//     Term 27 (AT2000-0250)/CC Outputs/Current setpoint value Ch.11 <-> Data Pointer/CurrentSetpointValues[10]
//     Term 27 (AT2000-0250)/CC Outputs/Current setpoint value Ch.12 <-> Data Pointer/CurrentSetpointValues[11]
//     Term 27 (AT2000-0250)/CC Outputs/Current setpoint value Ch.13 <-> Data Pointer/CurrentSetpointValues[12]
//     Term 27 (AT2000-0250)/CC Outputs/Current setpoint value Ch.14 <-> Data Pointer/CurrentSetpointValues[13]
//     Term 27 (AT2000-0250)/CC Outputs/Current setpoint value Ch.15 <-> Data Pointer/CurrentSetpointValues[14]
//     Term 27 (AT2000-0250)/CC Outputs/Current setpoint value Ch.2 <-> Data Pointer/CurrentSetpointValues[1]
//     Term 27 (AT2000-0250)/CC Outputs/Current setpoint value Ch.3 <-> Data Pointer/CurrentSetpointValues[2]
//     Term 27 (AT2000-0250)/CC Outputs/Current setpoint value Ch.4 <-> Data Pointer/CurrentSetpointValues[3]
//     Term 27 (AT2000-0250)/CC Outputs/Current setpoint value Ch.5 <-> Data Pointer/CurrentSetpointValues[4]
//     Term 27 (AT2000-0250)/CC Outputs/Current setpoint value Ch.6 <-> Data Pointer/CurrentSetpointValues[5]
//     Term 27 (AT2000-0250)/CC Outputs/Current setpoint value Ch.7 <-> Data Pointer/CurrentSetpointValues[6]
//     Term 27 (AT2000-0250)/CC Outputs/Current setpoint value Ch.8 <-> Data Pointer/CurrentSetpointValues[7]
//     Term 27 (AT2000-0250)/CC Outputs/Current setpoint value Ch.9 <-> Data Pointer/CurrentSetpointValues[8]
//     Term 27 (AT2000-0250)/Term 28 (AT2000-5250)/FB Inputs/Value Channel 01 <-> Data Pointer/RawPositionValues[0]
//     Term 27 (AT2000-0250)/Term 28 (AT2000-5250)/FB Inputs/Value Channel 02 <-> Data Pointer/RawPositionValues[1]
//     Term 27 (AT2000-0250)/Term 28 (AT2000-5250)/FB Inputs/Value Channel 03 <-> Data Pointer/RawPositionValues[2]
//     Term 27 (AT2000-0250)/Term 28 (AT2000-5250)/FB Inputs/Value Channel 04 <-> Data Pointer/RawPositionValues[3]
//     Term 27 (AT2000-0250)/Term 28 (AT2000-5250)/FB Inputs/Value Channel 05 <-> Data Pointer/RawPositionValues[4]
//     Term 27 (AT2000-0250)/Term 28 (AT2000-5250)/FB Inputs/Value Channel 06 <-> Data Pointer/RawPositionValues[5]
//     Term 27 (AT2000-0250)/Term 28 (AT2000-5250)/FB Inputs/Value Channel 07 <-> Data Pointer/RawPositionValues[6]
//     Term 27 (AT2000-0250)/Term 28 (AT2000-5250)/FB Inputs/Value Channel 08 <-> Data Pointer/RawPositionValues[7]
//     Term 27 (AT2000-0250)/Term 28 (AT2000-5250)/FB Inputs/Value Channel 09 <-> Data Pointer/RawPositionValues[8]
//     Term 27 (AT2000-0250)/Term 28 (AT2000-5250)/FB Inputs/Value Channel 10 <-> Data Pointer/RawPositionValues[9]
//     Term 27 (AT2000-0250)/Term 28 (AT2000-5250)/FB Inputs/Value Channel 11 <-> Data Pointer/RawPositionValues[10]
//     Term 27 (AT2000-0250)/Term 28 (AT2000-5250)/FB Inputs/Value Channel 12 <-> Data Pointer/RawPositionValues[11]
//     Term 27 (AT2000-0250)/Term 28 (AT2000-5250)/FB Inputs/Value Channel 13 <-> Data Pointer/RawPositionValues[12]
//     Term 27 (AT2000-0250)/Term 28 (AT2000-5250)/FB Inputs/Value Channel 14 <-> Data Pointer/RawPositionValues[13]
//     Term 27 (AT2000-0250)/Term 28 (AT2000-5250)/FB Inputs/Value Channel 15 <-> Data Pointer/RawPositionValues[14]
//     Term 27 (AT2000-0250)/Term 28 (AT2000-5250)/FB Inputs/Value Channel 16 <-> Data Pointer/RawPositionValues[15]
//     Term 27 (AT2000-0250)/Term 28 (AT2000-5250)/FB Inputs/Value Channel 17 <-> Data Pointer/RawPositionValues[16]
//     Term 27 (AT2000-0250)/Term 28 (AT2000-5250)/FB Inputs/Value Channel 18 <-> Data Pointer/RawPositionValues[17]
//     Term 27 (AT2000-0250)/Term 28 (AT2000-5250)/FB Inputs/Value Channel 19 <-> Data Pointer/RawPositionValues[18]
//     Term 27 (AT2000-0250)/Term 28 (AT2000-5250)/FB Inputs/Value Channel 20 <-> Data Pointer/RawPositionValues[19]
//     Term 27 (AT2000-0250)/Term 28 (AT2000-5250)/FB Inputs/Value Channel 21 <-> Data Pointer/RawPositionValues[20]
//     Term 27 (AT2000-0250)/Term 28 (AT2000-5250)/FB Inputs/Value Channel 22 <-> Data Pointer/RawPositionValues[21]
//     Term 27 (AT2000-0250)/Term 28 (AT2000-5250)/FB Inputs/Value Channel 23 <-> Data Pointer/RawPositionValues[22]
//     Term 27 (AT2000-0250)/Term 28 (AT2000-5250)/FB Inputs/Value Channel 24 <-> Data Pointer/RawPositionValues[23]
//     Term 27 (AT2000-0250)/Term 28 (AT2000-5250)/FB Inputs/Value Channel 25 <-> Data Pointer/RawPositionValues[24]
//     Term 27 (AT2000-0250)/Term 28 (AT2000-5250)/FB Inputs/Value Channel 26 <-> Data Pointer/RawPositionValues[25]
//     Term 27 (AT2000-0250)/Term 28 (AT2000-5250)/FB Inputs/Value Channel 27 <-> Data Pointer/RawPositionValues[26]
//     Term 27 (AT2000-0250)/Term 28 (AT2000-5250)/FB Inputs/Value Channel 28 <-> Data Pointer/RawPositionValues[27]
//     Term 27 (AT2000-0250)/Term 28 (AT2000-5250)/FB Inputs/Value Channel 29 <-> Data Pointer/RawPositionValues[28]
//     Term 27 (AT2000-0250)/Term 28 (AT2000-5250)/FB Inputs/Value Channel 30 <-> Data Pointer/RawPositionValues[29]
//     Term 27 (AT2000-0250)/Term 28 (AT2000-5250)/FB Inputs/Value Channel 31 <-> Data Pointer/RawPositionValues[30]
//     Term 27 (AT2000-0250)/Term 28 (AT2000-5250)/FB Inputs/Value Channel 32 <-> Data Pointer/RawPositionValues[31]
//   PLC1/PLC1 Instance <-> NC SAF/Axes/Mover Axis 1
//     PlcTask Inputs/MAIN.XTS.Mover[1].AxisReference.NcToPlc <-> Outputs/ToPlc
//     PlcTask Outputs/MAIN.XTS.Mover[1].AxisReference.PlcToNc <-> Inputs/FromPlc
//   PLC1/PLC1 Instance <-> NC SAF/Axes/Mover Axis 10
//     PlcTask Inputs/MAIN.XTS.Mover[10].AxisReference.NcToPlc <-> Outputs/ToPlc
//     PlcTask Outputs/MAIN.XTS.Mover[10].AxisReference.PlcToNc <-> Inputs/FromPlc
//   PLC1/PLC1 Instance <-> NC SAF/Axes/Mover Axis 2
//     PlcTask Inputs/MAIN.XTS.Mover[2].AxisReference.NcToPlc <-> Outputs/ToPlc
//     PlcTask Outputs/MAIN.XTS.Mover[2].AxisReference.PlcToNc <-> Inputs/FromPlc
//   PLC1/PLC1 Instance <-> NC SAF/Axes/Mover Axis 3
//     PlcTask Inputs/MAIN.XTS.Mover[3].AxisReference.NcToPlc <-> Outputs/ToPlc
//     PlcTask Outputs/MAIN.XTS.Mover[3].AxisReference.PlcToNc <-> Inputs/FromPlc
//   PLC1/PLC1 Instance <-> NC SAF/Axes/Mover Axis 4
//     PlcTask Inputs/MAIN.XTS.Mover[4].AxisReference.NcToPlc <-> Outputs/ToPlc
//     PlcTask Outputs/MAIN.XTS.Mover[4].AxisReference.PlcToNc <-> Inputs/FromPlc
//   PLC1/PLC1 Instance <-> NC SAF/Axes/Mover Axis 5
//     PlcTask Inputs/MAIN.XTS.Mover[5].AxisReference.NcToPlc <-> Outputs/ToPlc
//     PlcTask Outputs/MAIN.XTS.Mover[5].AxisReference.PlcToNc <-> Inputs/FromPlc
//   PLC1/PLC1 Instance <-> NC SAF/Axes/Mover Axis 6
//     PlcTask Inputs/MAIN.XTS.Mover[6].AxisReference.NcToPlc <-> Outputs/ToPlc
//     PlcTask Outputs/MAIN.XTS.Mover[6].AxisReference.PlcToNc <-> Inputs/FromPlc
//   PLC1/PLC1 Instance <-> NC SAF/Axes/Mover Axis 7
//     PlcTask Inputs/MAIN.XTS.Mover[7].AxisReference.NcToPlc <-> Outputs/ToPlc
//     PlcTask Outputs/MAIN.XTS.Mover[7].AxisReference.PlcToNc <-> Inputs/FromPlc
//   PLC1/PLC1 Instance <-> NC SAF/Axes/Mover Axis 8
//     PlcTask Inputs/MAIN.XTS.Mover[8].AxisReference.NcToPlc <-> Outputs/ToPlc
//     PlcTask Outputs/MAIN.XTS.Mover[8].AxisReference.PlcToNc <-> Inputs/FromPlc
//   PLC1/PLC1 Instance <-> NC SAF/Axes/Mover Axis 9
//     PlcTask Inputs/MAIN.XTS.Mover[9].AxisReference.NcToPlc <-> Outputs/ToPlc
//     PlcTask Outputs/MAIN.XTS.Mover[9].AxisReference.PlcToNc <-> Inputs/FromPlc
//   PLC1/PLC1 Instance <-> NC SAF/Objects/Collision Avoidance
//     PlcTask Inputs/MAIN.XTS.System.GROUP_REF.NcToPlc/CA <-> Group Outputs/ToPLC
//     PlcTask Outputs/MAIN.XTS.System.GROUP_REF.PlcToNc/CA <-> Group Inputs/FromPLC

CONFIGURATION PLC1
    RESOURCE PLC ON TwinCAT3
        TASK PLC_Slow(INTERVAL := T#100000us, PRIORITY := 20);
        PROGRAM HMIHelper WITH PLC_Slow : HMIHelper;
        PROGRAM DiagnosticPRG WITH PLC_Slow : DiagnosticPRG;
    END_RESOURCE
END_CONFIGURATION

// ---- DUTs/HMI_XTSMoverInfo_typ.TcDUT
TYPE HMI_XTSMoverInfo_typ :
STRUCT
	Index		: UDINT;
	Ready		: BOOL;
	Position	: LREAL;
END_STRUCT
END_TYPE

// ---- POUs/Diagnostics/XTSDiag/XTSDiag_InfeedSectionInfo.TcDUT
TYPE XTSDiag_InfeedSectionInfo :
STRUCT
	DcLinkVoltage				: ARRAY[1..6] OF REAL;
	ModuleCurrentSummed			: ARRAY[1..6] OF REAL;
	ModuleCurrentIndivual		: ARRAY[1..6] OF REAL;
	MaxOverallCurrentLast500ms	: ARRAY[1..6] OF REAL;
	ModuleNumber				: ARRAY[1..6] OF UDINT;
	ModuleCount					: INT;
	StartDcLinkVoltage			: REAL;
	EndDcLinkVoltage			: REAL;
	VoltageDropAcrossInfeed		: REAL;
	VoltageDropAcrossCable		: REAL;
	TotalCurrent				: REAL;
END_STRUCT
END_TYPE

// ---- POUs/Diagnostics/XTSDiag/XTSDiag_ModuleInfeedMapping_typ.TcDUT
TYPE XTSDiag_ModuleInfeedMapping_typ :
STRUCT
	Infeed		: INT;
	Position	: INT;
END_STRUCT
END_TYPE

// ---- POUs/Diagnostics/XTSDiag/XTSDiag_ModuleInfo.TcDUT
TYPE XTSDiag_ModuleInfo :
STRUCT
	DCLinkVoltage				: ARRAY[1..GVL_XTSDiag.MAX_NUM_MODULES] OF REAL;
	OverallCurrent				: ARRAY[1..GVL_XTSDiag.MAX_NUM_MODULES] OF REAL;
	MaxOverallCurrentLast500ms	: ARRAY[1..GVL_XTSDiag.MAX_NUM_MODULES] OF REAL;
	PCBTemperatures				: ARRAY[1..GVL_XTSDiag.MAX_NUM_MODULES] OF ARRAY[1..4] OF REAL;
	I2TTemperaturesPct			: ARRAY[1..GVL_XTSDiag.MAX_NUM_MODULES] OF ARRAY[1..15] OF USINT;
END_STRUCT
END_TYPE

// ---- POUs/Diagnostics/XTSDiag/XTSDiag_ModuleInfo_ByObj.TcDUT
TYPE XTSDiag_ModuleInfo_ByObj :
STRUCT
	DCLinkVoltage				: REAL;
	OverallCurrent				: REAL;
	MaxOverallCurrentLast500ms	: REAL;
	PCBTemperatures				: ARRAY[1..4] OF REAL;
	I2TTemperaturesPct			: ARRAY[1..15] OF USINT;
END_STRUCT
END_TYPE

// ---- POUs/Diagnostics/XTSDiag/XTSDiag_MoverInfo.TcDUT
TYPE XTSDiag_MoverInfo :
STRUCT
	FollowingError	: ARRAY[1..GVL_XTSDiag.MAX_NUM_MOVERS] OF LREAL;
	SetPosition		: ARRAY[1..GVL_XTSDiag.MAX_NUM_MOVERS] OF LREAL;
	SetVelocity		: ARRAY[1..GVL_XTSDiag.MAX_NUM_MOVERS] OF REAL;
	SetAcceleration	: ARRAY[1..GVL_XTSDiag.MAX_NUM_MOVERS] OF REAL;
	SetCurrent		: ARRAY[1..GVL_XTSDiag.MAX_NUM_MOVERS] OF LREAL;
	SetForce		: ARRAY[1..GVL_XTSDiag.MAX_NUM_MOVERS] OF LREAL;
	Error			: ARRAY[1..GVL_XTSDiag.MAX_NUM_MOVERS] OF BOOL;
	ErrorID			: ARRAY[1..GVL_XTSDiag.MAX_NUM_MOVERS] OF UDINT;
	Ready			: ARRAY[1..GVL_XTSDiag.MAX_NUM_MOVERS] OF BOOL;
END_STRUCT
END_TYPE

// ---- POUs/Diagnostics/XTSDiag/XTSDiag_MoverInfo_ByObj.TcDUT
TYPE XTSDiag_MoverInfo_ByObj :
STRUCT
	FollowingError	: LREAL;
	SetPosition		: LREAL;
	SetVelocity		: REAL;
	SetAcceleration	: REAL;
	SetCurrent		: LREAL;
	SetForce		: LREAL;
	Error			: BOOL;
	ErrorID			: UDINT;
	Ready			: BOOL;
END_STRUCT
END_TYPE

// ---- POUs/Diagnostics/XTSDiag/XTSDiag_SystemInfo.TcDUT
TYPE XTSDiag_SystemInfo :
STRUCT
	BusVoltage			: ARRAY[0..1] OF REAL;	
	ModuleCount			: UDINT;
	MoverCount			: UDINT;
	TotalMoverCurrent	: REAL;	// Sum of Mover Set Currents
	TotalModuleCurrent	: REAL; // Sum of Motor Overall Currents
	AvailableContinuousCurrent	: REAL;

	TotalCurrentUsagePct_MoverCalc	: REAL;	// TotalMoverCurrent divided by available current
	TotalCurrentUsagePct_ModuleCalc	: REAL;	// TotalModuleCurrent divided by available current
END_STRUCT
END_TYPE

// ---- XtsNctBaseUnit/DUTs/ST_NctProcessData.TcDUT
TYPE ST_NctProcessData :
STRUCT
	///Process data
	AppData0: USINT;
	AppData1: USINT;
	AppData2: USINT;
	AppData3: USINT;
	AppData4: USINT;
END_STRUCT
END_TYPE

// ---- XtsNctBaseUnit/DUTs/ST_NctProcessImage.TcDUT
TYPE ST_NctProcessImage :
STRUCT
	DigitalInput11	: BOOL;		//Bit
	DigitalInput12	: BOOL;		//Bit
	DigitalInput13	: BOOL;		//Bit
	DigitalInput14	: BOOL;		//Bit
	DigitalOutput11	: BOOL;		//Bit
	DigitalOutput12	: BOOL;		//Bit
	DigitalOutput13	: BOOL;		//Bit
	DigitalOutput14	: BOOL;		//Bit
	AnalogInput1	: LREAL;	//0-10V
	AnalogInput2	: LREAL;	//0-10V
	PwmFrequnecy	: LREAL;	//32kHz-128kHz
	PwmChannel1		: LREAL;	//0-100%
	PwmChannel2		: LREAL;	//0-100%
	PwmChannel3		: LREAL;	//0-100%
END_STRUCT
END_TYPE

// ---- XtsNctBaseUnit/DUTs/ST_NctRegisters.TcDUT
TYPE ST_NctRegisters :
STRUCT
	AdcCalibration			: ARRAY [1..32] OF BYTE;
	AdcCalibrationChannel3	: ARRAY [1..8] 	OF BYTE;
	AdcCalibrationChannel4	: ARRAY [1..8] 	OF BYTE;
	AdcInputChannel3		: INT;
	AdcInputChannel4		: INT;
	AdcRawInputChannel3		: INT;
	AdcRawInputChannel4		: INT;
	AntennaValues			: ARRAY [1..4] 	OF BYTE;
	ApplicationVersion		: STRING(31);
	Bic						: ARRAY [1..256] OF BYTE;
	BootloaderVersion		: STRING(31);
	Codeword				: UDINT;
	CommunicationVersion	: STRING(31);
	ControlVoltage			: UINT;
	DeviceId				: UDINT;
	DeviceName				: STRING(31);
	DiagHistoryBuffer		: ARRAY [1..256] OF BYTE;
	DiagHistoryControl		: USINT;
	DiagHistoryStatus		: USINT;
	DiagInfo				: UINT;
	HardwareVersion			: STRING(31);
	Identity				: ProductIdentity;
	MoverGuid				: GUID;
	MoverUsername			: STRING(31);
	RfidSettings			: ARRAY [1..4] 	OF BYTE;
	LocalAddress			: USINT;
	SoftwareVersion			: STRING(31);
	StackVersion			: STRING(31);
	SupplyCurrrent			: UINT;
	SupplyVoltage			: UINT;
	UserData				: ARRAY [1..32] OF BYTE;
	UserDataEE				: ARRAY [1..32] OF BYTE;
END_STRUCT
END_TYPE

// ---- XtsNctBaseUnit/DUTs/ST_ReturnStructure.TcDUT
TYPE ST_ReturnStructure :
STRUCT
	Done	: BOOL;
	Active	: BOOL;
	Busy	: BOOL;
	Aborted	: BOOL;
	Error	: BOOL;
	ErrorId	: UDINT;
END_STRUCT
END_TYPE

// ---- GVLs/Param.TcGVL
{attribute 'qualified_only'}
VAR_GLOBAL CONSTANT
	// The following should be set to a value **equal to or greater than** the number of movers needed
	MAX_MOVERS   			: USINT := 100;   // Movers
	
	// The following should be set to a value **equal to or greater than** the number of objectives needed
	NUM_MOVERLISTS			: USINT := 10;	// Mover Lists
	NUM_POSITIONTRIGGERS	: USINT := 10;	// Position Triggers
	NUM_STATIONS			: USINT := 10;	// Stations
	NUM_ZONES				: USINT := 10;	// Zones
	
	NUM_TRACKS				: USINT	:= 1;	// Tracks (Typically 1)
	DEFAULT_TRACK			: USINT := 0;	// Default track for movers, stations, zones and position triggers

	PART_ARRAY_SIZE			: UDINT := 100;
	AUTO_POPULATE_STATIONS  : BOOL := TRUE; // use the Station[x] array to label stations on the visualization. Turn off if manually entering stations in the configurator.

	// statistics weighted average
	ALPHA_EMA				: LREAL := 0.1;
END_VAR

// ---- POUs/Diagnostics/XTSDiag/GVL_XTSDiag.TcGVL
{attribute 'qualified_only'}
VAR_GLOBAL CONSTANT
	MAX_NUM_MOVERS	: UDINT	:= 10;
	MAX_NUM_MODULES	: UDINT	:= 12;
	MAX_NUM_INFEEDS	: UDINT	:= 2;
END_VAR

// ---- XtsNctBaseUnit/ITF/I_XtsNctBaseUnit.TcIO
INTERFACE I_XtsNctBaseUnit

{attribute 'monitoring' := 'call'}
PROPERTY ActiveTime : REAL
GET
END_GET
END_PROPERTY

{attribute 'monitoring' := 'call'}
PROPERTY AnalogInput1 : LREAL
GET
END_GET
END_PROPERTY

{attribute 'monitoring' := 'call'}
PROPERTY AnalogInput2 : LREAL
GET
END_GET
END_PROPERTY

PROPERTY BIC : ARRAY[1..256] OF BYTE
GET
END_GET
SET
END_SET
END_PROPERTY

{attribute 'monitoring' := 'call'}
PROPERTY ControlVoltage : UINT
GET
END_GET
SET
END_SET
END_PROPERTY

{attribute 'monitoring' := 'call'}
PROPERTY DeviceName : STRING(31)
GET
END_GET
SET
END_SET
END_PROPERTY

{attribute 'monitoring' := 'call'}
PROPERTY DigitalInput1 : BOOL
GET
END_GET
END_PROPERTY

{attribute 'monitoring' := 'call'}
PROPERTY DigitalInput2 : BOOL
GET
END_GET
END_PROPERTY

{attribute 'monitoring' := 'call'}
PROPERTY DigitalInput3 : BOOL
GET
END_GET
END_PROPERTY

{attribute 'monitoring' := 'call'}
PROPERTY DigitalInput4 : BOOL
GET
END_GET
END_PROPERTY

{attribute 'monitoring' := 'call'}
PROPERTY DigitalOutput1 : BOOL
GET
END_GET
SET
END_SET
END_PROPERTY

{attribute 'monitoring' := 'call'}
PROPERTY DigitalOutput2 : BOOL
GET
END_GET
SET
END_SET
END_PROPERTY

{attribute 'monitoring' := 'call'}
PROPERTY DigitalOutput3 : BOOL
GET
END_GET
SET
END_SET
END_PROPERTY

{attribute 'monitoring' := 'call'}
PROPERTY DigitalOutput4 : BOOL
GET
END_GET
SET
END_SET
END_PROPERTY

{attribute 'monitoring' := 'call'}
PROPERTY HardwareVersion : STRING(3)
GET
END_GET
SET
END_SET
END_PROPERTY

{attribute 'monitoring' := 'call'}
PROPERTY Identity : REFERENCE TO ProductIdentity
GET
END_GET
SET
END_SET
END_PROPERTY

METHOD Initalize : REFERENCE TO ST_ReturnStructure

VAR_INPUT
	bExecute: BOOL;
END_VAR
END_METHOD

{attribute 'monitoring' := 'call'}
PROPERTY InputProcessData : REFERENCE TO ST_NctProcessData
GET
END_GET
END_PROPERTY

{attribute 'monitoring' := 'call'}
PROPERTY IsInterfaceAssigned : BOOL
GET
END_GET
END_PROPERTY

PROPERTY MoverGuid : GUID
GET
END_GET
SET
END_SET
END_PROPERTY

{attribute 'monitoring' := 'call'}
PROPERTY MoverUsername : STRING(31)
GET
END_GET
SET
END_SET
END_PROPERTY

PROPERTY NctBaseUnitInterface : I_TcIoXtsNctBaseUnitInterface
GET
END_GET
END_PROPERTY

{attribute 'monitoring' := 'call'}
PROPERTY OutputProcessData : REFERENCE TO ST_NctProcessData
GET
END_GET
SET
END_SET
END_PROPERTY

{attribute 'monitoring' := 'call'}
PROPERTY PwmChannel1 : LREAL
GET
END_GET
SET
END_SET
END_PROPERTY

{attribute 'monitoring' := 'call'}
PROPERTY PwmChannel2 : LREAL
GET
END_GET
SET
END_SET
END_PROPERTY

{attribute 'monitoring' := 'call'}
PROPERTY PwmChannel3 : LREAL
GET
END_GET
SET
END_SET
END_PROPERTY

{attribute 'monitoring' := 'call'}
PROPERTY PwmFrequency : LREAL
GET
END_GET
SET
END_SET
END_PROPERTY

METHOD ReadRegister : REFERENCE TO ST_ReturnStructure

VAR_INPUT
	bExecute		: BOOL;
	stRegisterType	: NctRegisterType;
END_VAR
END_METHOD

{attribute 'monitoring' := 'call'}
PROPERTY Status : REFERENCE TO NctBaseUnitStatus
GET
END_GET
END_PROPERTY

METHOD UpdateProcessData : REFERENCE TO ST_ReturnStructure

VAR_INPUT
	bEnable	: BOOL;	//Enables the cylcilc communication
END_VAR
END_METHOD

METHOD WriteRegister : REFERENCE TO ST_ReturnStructure

VAR_INPUT
	bExecute		: BOOL;
	stRegisterType	: NctRegisterType;
END_VAR
END_METHOD

END_INTERFACE

// ---- POUs/HMIHelper.TcPOU
PROGRAM HMIHelper
VAR
	HMI_XTSMoverInfo	: ARRAY[1..10] OF HMI_XTSMoverInfo_typ;
	i					: INT;
	Init				: BOOL;
END_VAR

IF NOT Init THEN
	FOR i := 1 TO (SIZEOF(HMI_XTSMoverInfo) / SIZEOF(HMI_XTSMoverInfo[1])) DO
		HMI_XTSMoverInfo[i].Index	:= i;
	END_FOR
	Init	:= TRUE;
END_IF

FOR i := 1 TO (SIZEOF(HMI_XTSMoverInfo) / SIZEOF(HMI_XTSMoverInfo[1])) DO
	HMI_XTSMoverInfo[i].Ready		:= Main.XTS.Mover[i].Ready;
	HMI_XTSMoverInfo[i].Position	:= Main.XTS.Mover[i].TrackInfo.TrackPosition;
END_FOR

END_PROGRAM

// ---- POUs/MAIN.TcPOU
PROGRAM MAIN
VAR	
	// declare XTS with <number of movers>
	XTS				: FB_XTS<10>;
	NCT_Mover		: ARRAY[1..10] OF FB_XtsNctBaseUnit;
	ipNCT_Mover		: ARRAY[1..10] OF I_TcIoXtsNctBaseUnitInterface;
	i				: INT;
	// Machine
	State			: MachineState_enum;

	// ========= Example Application Variables =========

    nextStation 			: USINT := 4;
                    	
	StationTimer 			: ARRAY[0..Param.NUM_STATIONS] OF TON; // timer blocks, for station dwells
	RecoveryComplete		: BOOL;
	
	Trig0MoverIndex			: UDINT;
	Trig0MoverPosLag		: LREAL;

END_VAR


(* ======================================================================================

--- XTS Starter Project ---

This MAIN (PRG) is intended to serve as an example, which can be modified to suit your specific application.

No programming changes should be necessary inside the provided XTS objects / function block definitions.
They are intended to be simply instantiated and controlled via the provided methods and properties.
However the objects are provided as open-source for modification and extension as needed.

Documentation for these objects can be found online at:
https://beckhoff-usa-community.github.io/XTS_Base/

Bug reports, new feature requests, and general feedback is always welcome on our Github page.
For any other questions, please reach out to your local Application Engineer.

- XTS Application Group | Beckhoff USA

====================================================================================== *)

(*
All sample code provided by Beckhoff Automation LLC are for illustrative purposes only
and are provided “as is” and without any warranties, express or implied. Actual
implementations in applications will vary significantly. Beckhoff Automation LLC shall
have no liability for, and does not waive any rights in relation to, any code samples that it
provides or the use of such code samples for any purpose.
*)

// main state machine
CASE State OF 

	// off (idle) state, waiting for enable command
	MS_OFF:
		// wait for enable command
		IF MainCommands.Enable THEN
			// initialize stations, positions and triggers
			Initializing();
			// enable the XTS
			XTS.Enable				:= TRUE;
			State					:= MS_RESTARTING;
		END_IF
		
	MS_RESTARTING:
		// restart the system by enabling the XTS and waiting for it to complete
		IF NOT MainCommands.Enable THEN
			// disable triggered, pass to xts and stop the movers
			XTS.Enable				:= FALSE;
			State					:= MS_STOPPED;
		ELSIF XTS.State = XTS_ENABLED THEN
			// enable complete move to enabled
			State		:= MS_ENABLED;
		END_IF


	MS_ENABLED:
		// XTS is enabled, wait for start command
		IF NOT MainCommands.Enable THEN
			XTS.Enable				:= FALSE;
			State					:= MS_STOPPED;
		ELSIF MainCommands.Start THEN
			// reset the recovery complete flag
			RecoveryComplete		:= FALSE;
			// move to next state
			State					:= MS_ONESHOT_RECOVER;
		END_IF
		
	MS_ONESHOT_RECOVER:
		// one time commands before starting typical process motions
		RecoverOneshot();
		State := MS_RECOVERING;
		
	MS_RECOVERING:
		// wait for any recovery actions to complete
		Recovering();
		// test for errors, commands or recovery complete
		IF MainCommands.Stop THEN
			// respond to stop command
			MainCommands.Start		:= FALSE;
			XTS.System.CompleteMoverList.HaltAll();
            State         	:= MS_STOPPED;
        ELSIF NOT MainCommands.Enable THEN
			// respond to loss of enable
            XTS.Enable		:= FALSE;
			XTS.System.CompleteMoverList.HaltAll();
            State          			:= MS_STOPPED;
		ELSIF RecoveryComplete THEN
			// recovery sequence is complete, move on to run state
			State					:= MS_RUNNING;
        END_IF

	MS_RUNNING:
		// run the station-to-station mover logic
		StationLogic();
		
		// monitor for disable or stop
		IF NOT MainCommands.Enable THEN
			XTS.Enable				:= FALSE;
			XTS.System.CompleteMoverList.HaltAll();
			State					:= MS_STOPPED;
		ELSIF MainCommands.Stop THEN
			MainCommands.Start		:= FALSE;
			XTS.System.CompleteMoverList.HaltAll();
			State					:= MS_STOPPED;
		END_IF

	MS_STOPPED:
		// movers are stopped, but XTS is still enabled
		// wait for restart, disable or error disable
		IF XTS.State <> XTS_ENABLED AND MainCommands.Enable THEN
			State					:= MS_ERROR;
		ELSIF NOT MainCommands.Enable THEN
			XTS.Enable 				:= FALSE;
		ELSIF  MainCommands.Start THEN
			MainCommands.Stop		:= FALSE;
			State					:= MS_ONESHOT_RECOVER;
		END_IF
		IF XTS.State = XTS_DISABLED THEN
			State					:= MS_OFF;
		END_IF;
	
END_CASE

// call the main XTS logic
XTS.CyclicLogic();


// NCT Control
(*FOR i := 9 TO 10 DO
	IF NCT_Mover[i].Status.isInitialized THEN
		NCT_Mover[i].UpdateProcessData(TRUE);
	END_IF
END_FOR	*)

ACTION Initializing:
// XTS Object Init
XTS.Station[0].Position 		:= 250;
XTS.Station[1].Position 		:= 750;
XTS.Station[2].Position 		:= 1750;
XTS.Station[3].Position 		:= 1850;
XTS.Station[4].Position 		:= 1950;

// station names
XTS.Station[0].Description		:= 'Load Top';
XTS.Station[1].Description		:= 'Load Bottom';
XTS.Station[2].Description		:= 'Weld A';
XTS.Station[3].Description		:= 'Weld B';
XTS.Station[4].Description		:= 'Weld C';

// speed changes in corners
XTS.PositionTrigger[0].Position := 1500;
XTS.PositionTrigger[1].Position := 2200;
XTS.PositionTrigger[2].Position := 2700;

// recover trigger near station 0
XTS.PositionTrigger[3].Position := XTS.Station[0].Position + 2.0;

// window around station 0 for startup
XTS.Zone[0].StartPosition		:= XTS.Station[0].Position - 1.0;
XTS.Zone[0].EndPosition   		:= XTS.Station[0].Position + 1.0;

XTS.InitialParameterSet.Velocity		:= 1000;		// mm/s
XTS.InitialParameterSet.Acceleration	:= 10_000;		// mm/s2
XTS.InitialParameterSet.Deceleration	:= 10_000;		// mm/s2
XTS.InitialParameterSet.Jerk			:= 100_000;		// mm/s3
XTS.InitialParameterSet.Gap				:= 95;			// mm
XTS.InitialParameterSet.Direction		:= Tc3_Mc3Definitions.MC_Direction.mcDirectionPositive;

MainCommands.lowVelocity	:= 300;
MainCommands.mediumVelocity	:= 800;
MainCommands.highVelocity	:= 1200;


//NCT
(*NCT_Mover[9].AssignInterface(ipNCT_Mover[9]);
NCT_Mover[10].AssignInterface(ipNCT_Mover[10]);

NCT_Mover[9].Initalize(TRUE);
NCT_Mover[10].Initalize(TRUE);		*)
END_ACTION

ACTION Recovering:
// this state is called until all movers have completed their desired recovery tasks

// wait for all movers to reach the standstill state and one mover at station 0
IF (XTS.System.CompleteMoverList.IsAllMoversHalted AND XTS.Station[0].MoverInPosition) THEN
	RecoveryComplete := TRUE;
END_IF

// position trigger leaving station 0 for recovery
IF XTS.PositionTrigger[3].MoverPassedPosition THEN
	XTS.PositionTrigger[3].CurrentMover.SetVelocity(MainCommands.mediumVelocity).MoveToStation(XTS.Station[0]);
	XTS.PositionTrigger[3].MuteCurrent();
END_IF
END_ACTION

ACTION RecoverOneshot:
// this action is called one time after the start command is issued
// it is intended to provide a single command to each mover to facilitate recovery
// other commands such as resetting counters and timers should also be carried out here

// send all movers to station 0
XTS.System.CompleteMoverList.SetAllVelocity(MainCommands.mediumVelocity).MoveAllToStation( XTS.Station[0] );
//movers near station 0 (zone 0) need to first move away from the station
XTS.Zone[0].CurrentMoverList.MoveAllVelocity(MainCommands.lowVelocity);
XTS.PositionTrigger[3].MuteCurrent();
// Restart statistics
XTS.System.ResetStatistics();

// Reinit nextStation
nextStation := 4;
END_ACTION

ACTION StationLogic:
		(*Mover routing logic should be written here to define the system's operating behavior.
		Station implementations, Position Trigger logic, etc. In general, you can remove the example code
		here down to the short line break that looks like this: // ============= *)
	
        // Station 0 Logic
        IF XTS.Station[0].MoverInPosition THEN
            StationTimer[0](IN := TRUE, PT := T#1000MS);
            IF StationTimer[0].Q THEN
                XTS.Mover[XTS.Station[0].CurrentMover.MoverIndex].MoveToStationByRampTime(
					DestinationStation:= XTS.Station[1], 
					Velocity:= 500, 
					RampTime:= 1.5, 
					Stiffness:= 0.5, 
					Gap:= 85);
            END_IF
        ELSE
            StationTimer[0](IN := FALSE);
        END_IF
		
        // Station 1 Logic		
        IF XTS.Station[1].MoverInPosition THEN
            StationTimer[1](IN := TRUE, PT := T#250MS);
            IF StationTimer[1].Q THEN
                XTS.Station[1].CurrentMover.MoveToStation(XTS.Station[nextStation]);
                nextStation := nextStation - 1;
                IF nextStation = 1 THEN
                    nextStation := 4;
                END_IF
            END_IF
        ELSE
            StationTimer[1](IN := FALSE);
        END_IF
		
		// Group of Stations 2, 3, and 4 Logic
        IF XTS.Station[2].MoverInPosition AND XTS.Station[3].MoverInPosition AND XTS.Station[4].MoverInPosition THEN
            StationTimer[2](IN := TRUE, PT := T#750MS);
            IF StationTimer[2].Q THEN
				StationTimer[2](IN := FALSE);
				
				XTS.Station[2].CurrentMover.MotionParameters:= XTS.InitialParameterSet;
				XTS.Station[3].CurrentMover.MotionParameters:= XTS.InitialParameterSet;
				XTS.Station[4].CurrentMover.MotionParameters:= XTS.InitialParameterSet;

                XTS.Station[2].CurrentMover.MoveVelocity(500);
                XTS.Station[3].CurrentMover.MoveVelocity(500);
                XTS.Station[4].CurrentMover.MoveVelocity(500);
				
            END_IF
        END_IF
		
        // Position Trigger 0 Logic
        IF XTS.PositionTrigger[0].MoverPassedPosition THEN
            XTS.PositionTrigger[0].CurrentMover.SetVelocity(MainCommands.lowVelocity);
			
			// To Call ApplicationMover addon Method/Properties/Variables, you must call Mover[] array index directly
			// Get MoverIndex for later use with ApplicationMover addons
			Trig0MoverIndex		:= XTS.PositionTrigger[0].CurrentMover.MoverIndex;
			
			// Call ApplicationMover Method/Properties/Variables using previously latched MoverIndex
			Trig0MoverPosLag	:= XTS.Mover[Trig0MoverIndex].PositionLag;
			
            XTS.PositionTrigger[0].MuteCurrent();
						
        END_IF
		
        // Position Trigger 1 Logic
        IF XTS.PositionTrigger[1].MoverPassedPosition THEN
			XTS.PositionTrigger[1].CurrentMover.SetAcceleration(5E2);
            XTS.PositionTrigger[1].CurrentMover.SetVelocity(MainCommands.highVelocity);
            XTS.PositionTrigger[1].MuteCurrent();
        END_IF

		// Position Trigger 2 Logic
        IF XTS.PositionTrigger[2].MoverPassedPosition THEN
			XTS.PositionTrigger[2].CurrentMover.SetAcceleration(1E4);
            XTS.PositionTrigger[2].CurrentMover.SetVelocity(MainCommands.lowVelocity);
            XTS.PositionTrigger[2].CurrentMover.MoveToStation(XTS.Station[0]);
            XTS.PositionTrigger[2].MuteCurrent();
        END_IF
END_ACTION

END_PROGRAM

// ---- XtsNctBaseUnit/POU/FB_XtsNctBaseUnit.TcPOU
FUNCTION_BLOCK FB_XtsNctBaseUnit IMPLEMENTS I_XtsNctBaseUnit

VAR
	//NCT Base Unit Interface interface
	_ipTcIoXtsNctBaseUnitInterface	: I_TcIoXtsNctBaseUnitInterface; //Reference to initalized XtsBaseUnitInteraface Function Block

	//ProcessData Input
	_stNctProcessDataIn		: ST_NctProcessData;
	
	//ProcessData Output
	_stNctProcessDataOut	: ST_NctProcessData;
	
	//Registers Output
	_aADCCalibration			: ARRAY[1..32] OF BYTE;
	_aADCCalibrationChannel3	: ARRAY[1..8] OF BYTE;
	_aADCCalibrationChannel4	: ARRAY[1..8] OF BYTE;
	_nADCInputChannel3			: INT;
	_nADCInputChannel4			: INT;
	_nADCRawInputChannel3		: INT;
	_nADCRawInputChannel4		: INT;
	_aAntennaValues				: ARRAY[1..4] OF BYTE;
	_aAny						: ARRAY[1..256] OF BYTE;
	_sApplicationVersion		: STRING(31);
	_aBIC						: ARRAY[1..256] OF BYTE;
	_sBootloaderVersion			: STRING(31);
	_nCodeword					: UDINT;
	_sCommunicationVersion		: STRING(31);
	_nControlVoltage			: UINT;
	_nDeviceId					: UDINT;
	_sDeviceName				: STRING(31);
	_aDiagHistoryBuffer			: ARRAY[1..256] OF BYTE;
	_nDiagHistoryControl		: USINT;
	_nDiagHistoryStatus			: USINT;
	_nDiagInfo					: UINT;
	_sHardwareVersion			: STRING(3);
	_stIdentity					: ProductIdentity;
	_nMTSHeaderSettings			: BYTE;
	_stMoverGuid				: GUID;
	_sMoverUsername				: STRING(31);
	_aRFIDSettings				: ARRAY[1..4] OF BYTE;
	_nLocalAddress				: USINT;
	_sSoftwareVersion			: STRING(31);
	_sStackVersion				: STRING(31);
	_nSupplyCurrent				: UINT;
	_nSupplyVoltage				: UINT;
	_aUserData					: ARRAY[1..32] OF BYTE;
	_aUserDataEE				: ARRAY[1..32] OF BYTE;
END_VAR

{attribute 'monitoring' := 'call'}
PROPERTY ActiveTime : REAL
GET
IF IsInterfaceAssigned THEN
	ActiveTime := _ipTcIoXtsNctBaseUnitInterface.GetActiveTime();
END_IF
END_GET
END_PROPERTY

{attribute 'monitoring' := 'call'}
PROPERTY AnalogInput1 : LREAL
GET
VAR
	nAnalogInput: UINT;
END_VAR
//Lowbyte
nAnalogInput.0 := _stNctProcessDataIn.AppData1.0;
nAnalogInput.1 := _stNctProcessDataIn.AppData1.1;
nAnalogInput.2 := _stNctProcessDataIn.AppData1.2;
nAnalogInput.3 := _stNctProcessDataIn.AppData1.3;
nAnalogInput.4 := _stNctProcessDataIn.AppData1.4;
nAnalogInput.5 := _stNctProcessDataIn.AppData1.5;
nAnalogInput.6 := _stNctProcessDataIn.AppData1.6;
nAnalogInput.7 := _stNctProcessDataIn.AppData1.7;

//Highbyte
nAnalogInput.8 	:= _stNctProcessDataIn.AppData2.0;
nAnalogInput.9 	:= _stNctProcessDataIn.AppData2.1;
nAnalogInput.10 := _stNctProcessDataIn.AppData2.2;
nAnalogInput.11 := _stNctProcessDataIn.AppData2.3;
nAnalogInput.12 := _stNctProcessDataIn.AppData2.4;
nAnalogInput.13 := _stNctProcessDataIn.AppData2.5;
nAnalogInput.14 := _stNctProcessDataIn.AppData2.6;
nAnalogInput.15 := _stNctProcessDataIn.AppData2.7;

//Convert to 10V scale
AnalogInput1:=(10.0/(4095)*nAnalogInput);
END_GET
END_PROPERTY

{attribute 'monitoring' := 'call'}
PROPERTY AnalogInput2 : LREAL
GET
VAR
	nAnalogInput: UINT;
END_VAR
//Lowbyte
nAnalogInput.0 := _stNctProcessDataIn.AppData3.0;
nAnalogInput.1 := _stNctProcessDataIn.AppData3.1;
nAnalogInput.2 := _stNctProcessDataIn.AppData3.2;
nAnalogInput.3 := _stNctProcessDataIn.AppData3.3;
nAnalogInput.4 := _stNctProcessDataIn.AppData3.4;
nAnalogInput.5 := _stNctProcessDataIn.AppData3.5;
nAnalogInput.6 := _stNctProcessDataIn.AppData3.6;
nAnalogInput.7 := _stNctProcessDataIn.AppData3.7;

//Highbyte
nAnalogInput.8 	:= _stNctProcessDataIn.AppData4.0;
nAnalogInput.9 	:= _stNctProcessDataIn.AppData4.1;
nAnalogInput.10 := _stNctProcessDataIn.AppData4.2;
nAnalogInput.11 := _stNctProcessDataIn.AppData4.3;
nAnalogInput.12 := _stNctProcessDataIn.AppData4.4;
nAnalogInput.13 := _stNctProcessDataIn.AppData4.5;
nAnalogInput.14 := _stNctProcessDataIn.AppData4.6;
nAnalogInput.15 := _stNctProcessDataIn.AppData4.7;

//Convert to 10V scale
AnalogInput2:=(10.0/4095)*(nAnalogInput);
END_GET
END_PROPERTY

METHOD AssignInterface : PVOID

VAR_INPUT
	ipTcIoXtsNctBaseUnitInterface	: I_TcIoXtsNctBaseUnitInterface;
END_VAR
//Nct Base Unit Interface-------------------------------------------------------------------
NctBaseUnitInterface	:= ipTcIoXtsNctBaseUnitInterface;
//Nct Base Unit Interface-------------------------------------------------------------------
END_METHOD

PROPERTY BIC : ARRAY[1..256] OF BYTE
GET
IF IsInterfaceAssigned THEN
	BIC := _ipTcIoXtsNctBaseUnitInterface.GetBIC();
END_IF
END_GET
SET
_aBIC	:= BIC;
END_SET
END_PROPERTY

{attribute 'monitoring' := 'call'}
PROPERTY ControlVoltage : UINT
GET
IF IsInterfaceAssigned THEN
	ControlVoltage := _ipTcIoXtsNctBaseUnitInterface.GetControlVoltage();
END_IF
END_GET
SET
_nControlVoltage	:= ControlVoltage;
END_SET
END_PROPERTY

{attribute 'monitoring' := 'call'}
PROPERTY DeviceName : STRING(31)
GET
IF IsInterfaceAssigned THEN
	DeviceName := _ipTcIoXtsNctBaseUnitInterface.GetDeviceName();
END_IF
END_GET
SET
_sDeviceName	:= DeviceName;
END_SET
END_PROPERTY

{attribute 'monitoring' := 'call'}
PROPERTY DigitalInput1 : BOOL
GET
DigitalInput1 := _stNctProcessDataIn.AppData0.0;
END_GET
END_PROPERTY

{attribute 'monitoring' := 'call'}
PROPERTY DigitalInput2 : BOOL
GET
DigitalInput2 := _stNctProcessDataIn.AppData0.1;
END_GET
END_PROPERTY

{attribute 'monitoring' := 'call'}
PROPERTY DigitalInput3 : BOOL
GET
DigitalInput3 := _stNctProcessDataIn.AppData0.2;
END_GET
END_PROPERTY

{attribute 'monitoring' := 'call'}
PROPERTY DigitalInput4 : BOOL
GET
DigitalInput4 := _stNctProcessDataIn.AppData0.3;
END_GET
END_PROPERTY

{attribute 'monitoring' := 'call'}
PROPERTY DigitalOutput1 : BOOL
GET
DigitalOutput1 := _stNctProcessDataOut.AppData0.0;
END_GET
SET
 _stNctProcessDataOut.AppData0.0:=DigitalOutput1;
END_SET
END_PROPERTY

{attribute 'monitoring' := 'call'}
PROPERTY DigitalOutput2 : BOOL
GET
DigitalOutput2 := _stNctProcessDataOut.AppData0.1;
END_GET
SET
_stNctProcessDataOut.AppData0.1:=DigitalOutput2;
END_SET
END_PROPERTY

{attribute 'monitoring' := 'call'}
PROPERTY DigitalOutput3 : BOOL
GET
DigitalOutput3 := _stNctProcessDataOut.AppData0.2;
END_GET
SET
_stNctProcessDataOut.AppData0.2:=DigitalOutput3;
END_SET
END_PROPERTY

{attribute 'monitoring' := 'call'}
PROPERTY DigitalOutput4 : BOOL
GET
DigitalOutput4 := _stNctProcessDataOut.AppData0.3;
END_GET
SET
_stNctProcessDataOut.AppData0.3:=DigitalOutput4;
END_SET
END_PROPERTY

{attribute 'monitoring' := 'call'}
PROPERTY HardwareVersion : STRING(3)
GET
IF IsInterfaceAssigned THEN
	HardwareVersion := _ipTcIoXtsNctBaseUnitInterface.GetHardwareVersion();
END_IF
END_GET
SET
_sHardwareVersion	:= HardwareVersion;
END_SET
END_PROPERTY

{attribute 'monitoring' := 'call'}
PROPERTY Identity : REFERENCE TO ProductIdentity
GET
IF IsInterfaceAssigned THEN
	Identity REF= _stIdentity;//_ipTcIoXtsNctBaseUnitInterface.GetIdentity();
END_IF
END_GET
SET
_stIdentity	:= Identity;
END_SET
END_PROPERTY

METHOD Initalize : REFERENCE TO ST_ReturnStructure

VAR_INPUT
	bExecute: BOOL;
END_VAR

VAR_OUTPUT
END_VAR

VAR_INST
	//Case
	nCase	: INT;
	
	//Return
	stReturnStructure	: ST_ReturnStructure;

	//Trigger
	fbRTrig: R_TRIG;
	fbFTrig: F_TRIG;

	//Command
	stNctCommandEntry	: NctCommandEntry;
	stNctCommandInfo	: NctCommandInfo;
	stNctCommandData	: ARRAY[1..256] OF BYTE;
	
	//Timeout	
	fbTimeout	: TON;
	
	//LogMessage
	aLogMessageThrown	: ARRAY[1..3] OF BOOL;
END_VAR	
	
VAR	
	//Command
	stNctInitCommandArguments	: NctInitCommandArguments;
	stAbortCommandArguments		: NctAbortCommandArguments;

	//Timeout
	tTimeoutTime	: TIME :=T#1S;	//Sets the time for timeout
	
	//LogMessage
	nNumLogMessages	: INT :=3;
	nForCounter		: INT;
END_VAR
fbRTrig(CLK:=bExecute);
fbFTrig(CLK:=bExecute);

//On rising Execute
IF fbRTrig.Q THEN
	//Update return
	stReturnStructure.Done		:= FALSE;
	stReturnStructure.Busy		:= TRUE;
	stReturnStructure.Active	:= FALSE;
	stReturnStructure.Aborted	:= FALSE;
	stReturnStructure.Error		:= FALSE;
	stReturnStructure.ErrorId	:= 0;
	
	//Set case
	nCase:=1;

//On falling Execute
ELSIF fbFTrig.Q THEN
	//Update return
	stReturnStructure.Done		:= FALSE;
	stReturnStructure.Busy		:= FALSE;
	stReturnStructure.Active	:= FALSE;
	stReturnStructure.Aborted	:= FALSE;
	stReturnStructure.Error		:= FALSE;
	stReturnStructure.ErrorId	:= 0;

	//Set case
	nCase:=0;
END_IF

CASE nCase OF
	0: //Idle
		;
	
	1: //Prepare Command
		IF Status.isMinActivationTimePassed AND Status.isReadyToInitialize THEN
		
			//Init Mode
			NctBaseUnitInterface.SetInitMode(NctInitMode.SimpleInit);
		
			//Command Parameters
			stNctInitCommandArguments.iterationCount 	:= 10;
			stNctInitCommandArguments.maxErrorCount 	:= 10;
			stNctInitCommandArguments.executionMode		:= NctCommandExecutionMode.UntilSuccessMaxErrors;
			
			//Add Write Init Command
			stNctCommandEntry	:= NctBaseUnitInterface.AddInitCommand(stNctInitCommandArguments);
			
			//Update return structure
			stReturnStructure.Done		:= FALSE;
			stReturnStructure.Busy		:= TRUE;
			stReturnStructure.Active	:= FALSE;
			stReturnStructure.Aborted	:= FALSE;
			stReturnStructure.Error		:= FALSE;
			stReturnStructure.ErrorId	:= 0;
			
			//Reset log messages
			FOR nForCounter:=1 TO nNumLogMessages DO
				aLogMessageThrown[nForCounter]	:= FALSE;
			END_FOR
			
			//Reset timeout timer
			fbTimeOut(IN:=FALSE);
			
			//Set case
			nCase:=2;
			
		ELSE
			//Update return structure
			stReturnStructure.Done		:= FALSE;
			stReturnStructure.Busy		:= FALSE;
			stReturnStructure.Active	:= FALSE;
			stReturnStructure.Aborted	:= FALSE;
			stReturnStructure.Error		:= TRUE;
			stReturnStructure.ErrorId	:= 1;
			
			//Write log message
			IF NOT aLogMessageThrown[stReturnStructure.ErrorId] THEN
				aLogMessageThrown[stReturnStructure.ErrorId]	:= TRUE;
				
				ADSLOGSTR(msgCtrlMask:=ADSLOG_MSGTYPE_ERROR ,msgFmtStr:='Initalizing %s not possible because the Base Unit is not ready to be initalized.',strArg:=NctBaseUnitInterface.P_ObjectName);
			END_IF
		
			//Set case
			nCase:=0;
		END_IF

	2: //Check Command
		stNctCommandInfo	:= NctBaseUnitInterface.GetCmdInfoByCmdEntry(stNctCommandEntry);
	
		IF 		stNctCommandInfo.status = NctCommandStatus.IsRunning THEN
			//Update return structure
			stReturnStructure.Done		:= FALSE;
			stReturnStructure.Busy		:= TRUE;
			stReturnStructure.Active	:= TRUE;
			stReturnStructure.Aborted	:= FALSE;
			stReturnStructure.Error		:= FALSE;
			stReturnStructure.ErrorId	:= 0;
			
			//Timeout
			fbTimeOut(IN:=TRUE, PT:=tTimeoutTime);
			
			IF fbTimeOut.Q THEN
				//Abort Command
				stAbortCommandArguments.option	:= NctAbortCommandParameterOption.ById;
				stAbortCommandArguments.id		:= stNctCommandEntry.id;
				NctBaseUnitInterface.AbortCommand(stAbortCommandArguments);
				
				//Update return structure
				stReturnStructure.Done		:= FALSE;
				stReturnStructure.Busy		:= FALSE;
				stReturnStructure.Active	:= FALSE;
				stReturnStructure.Aborted	:= FALSE;
				stReturnStructure.Error		:= TRUE;
				stReturnStructure.ErrorId	:= 3;
				
				//Write log message
				IF NOT aLogMessageThrown[stReturnStructure.ErrorId] THEN
					aLogMessageThrown[stReturnStructure.ErrorId]	:= TRUE;
					
					ADSLOGSTR(msgCtrlMask:=ADSLOG_MSGTYPE_ERROR ,msgFmtStr:='Initalizing %s not possible because the method went into timeout.',strArg:=NctBaseUnitInterface.P_ObjectName);
				END_IF
				
				//Next step
				nCase:=0;
			END_IF
			
		ELSIF 	stNctCommandInfo.status = NctCommandStatus.IsQueued OR
				stNctCommandInfo.status = NctCommandStatus.IsWaitingForStartConditions OR
				stNctCommandInfo.status = NctCommandStatus.IsWaitingToResume THEN
				
			//Update return structure
			stReturnStructure.Done		:= FALSE;
			stReturnStructure.Busy		:= TRUE;
			stReturnStructure.Active	:= FALSE;
			stReturnStructure.Aborted	:= FALSE;
			stReturnStructure.Error		:= FALSE;
			stReturnStructure.ErrorId	:= 0;	
			
		ELSIF 	stNctCommandInfo.status = NctCommandStatus.IsSucceeded THEN
			stNctCommandData	:= NctBaseUnitInterface.GetCmdDataByCmdEntry(stNctCommandEntry);
			
			//Process Data
			_stNctProcessDataIn.AppData0	:= stNctCommandData[1];
			_stNctProcessDataIn.AppData1	:= stNctCommandData[2];
			_stNctProcessDataIn.AppData2	:= stNctCommandData[3];
			_stNctProcessDataIn.AppData3	:= stNctCommandData[4];
			_stNctProcessDataIn.AppData4	:= stNctCommandData[5];
			
			//Update return structure
			stReturnStructure.Done		:= TRUE;
			stReturnStructure.Busy		:= FALSE;
			stReturnStructure.Active	:= FALSE;
			stReturnStructure.Aborted	:= FALSE;
			stReturnStructure.Error		:= FALSE;
			stReturnStructure.ErrorId	:= 0;
		
			//Next step
			nCase:=0;
			
		ELSIF 	stNctCommandInfo.status = NctCommandStatus.IsAbortedByArea OR
				stNctCommandInfo.status = NctCommandStatus.IsAbortedByUser THEN
				
			//Update return structure
			stReturnStructure.Done		:= FALSE;
			stReturnStructure.Busy		:= FALSE;
			stReturnStructure.Active	:= FALSE;
			stReturnStructure.Aborted	:= TRUE;
			stReturnStructure.Error		:= FALSE;
			stReturnStructure.ErrorId	:= 0;	
				
			//Next step
			nCase:=0;
			
		ELSIF 	stNctCommandInfo.status = NctCommandStatus.IsFailed OR
				stNctCommandInfo.status = NctCommandStatus.IsFailedDueToChildCommand OR
				stNctCommandInfo.status = NctCommandStatus.IsInitFailedDueToCorruptedArgs OR
				stNctCommandInfo.status = NctCommandStatus.IsInitFailedDueToInvalidArgs OR
				stNctCommandInfo.status = NctCommandStatus.IsInitFailedDueToNoMemory OR
				stNctCommandInfo.status = NctCommandStatus.IsInitFailedDueToNotSupportedRegister THEN
				
			//Update return structure
			stReturnStructure.Done		:= FALSE;
			stReturnStructure.Busy		:= FALSE;
			stReturnStructure.Active	:= FALSE;
			stReturnStructure.Aborted	:= FALSE;
			stReturnStructure.Error		:= TRUE;
			stReturnStructure.ErrorId	:= 2;	
			
			//Write log message
			IF NOT aLogMessageThrown[stReturnStructure.ErrorId] THEN
				aLogMessageThrown[stReturnStructure.ErrorId]	:= TRUE;
				
				ADSLOGSTR(msgCtrlMask:=ADSLOG_MSGTYPE_ERROR ,msgFmtStr:='Initalizing %s not possible because command failed.',strArg:=NctBaseUnitInterface.P_ObjectName);
			END_IF
			
			//Next step
			nCase:=0;
			
		ELSIF	stNctCommandInfo.status = NctCommandStatus.NotDefined THEN
			;
		END_IF
			
END_CASE

//Update return structure
Initalize	REF= stReturnStructure;
END_METHOD

{attribute 'monitoring' := 'call'}
PROPERTY InputProcessData : REFERENCE TO ST_NctProcessData
GET
InputProcessData REF= _stNctProcessDataIn;
END_GET
END_PROPERTY

{attribute 'monitoring' := 'call'}
PROPERTY IsInterfaceAssigned : BOOL
GET
IF _ipTcIoXtsNctBaseUnitInterface <> 0 THEN
	IsInterfaceAssigned := TRUE;
END_IF
END_GET
END_PROPERTY

PROPERTY MoverGuid : GUID
GET
IF IsInterfaceAssigned THEN
	MoverGuid := _ipTcIoXtsNctBaseUnitInterface.GetMoverGuid();
END_IF
END_GET
SET
_stMoverGuid	:= MoverGuid;
END_SET
END_PROPERTY

{attribute 'monitoring' := 'call'}
PROPERTY MoverUsername : STRING(31)
GET
IF IsInterfaceAssigned THEN
	MoverUsername := _ipTcIoXtsNctBaseUnitInterface.GetMoverUsername();
END_IF
END_GET
SET
_sMoverUsername	:= MoverUsername;
END_SET
END_PROPERTY

PROPERTY NctBaseUnitInterface : I_TcIoXtsNctBaseUnitInterface
GET
NctBaseUnitInterface := _ipTcIoXtsNctBaseUnitInterface;
END_GET
SET
_ipTcIoXtsNctBaseUnitInterface	:= NctBaseUnitInterface;
END_SET
END_PROPERTY

{attribute 'monitoring' := 'call'}
PROPERTY OutputProcessData : REFERENCE TO ST_NctProcessData
GET
OutputProcessData	REF= _stNctProcessDataOut;
END_GET
SET
_stNctProcessDataOut	:= OutputProcessData;
END_SET
END_PROPERTY

{attribute 'monitoring' := 'call'}
PROPERTY PwmChannel1 : LREAL
GET
PwmChannel1	:= 100.0/255*_stNctProcessDataOut.AppData2;
END_GET
SET
_stNctProcessDataOut.AppData2	:= LREAL_TO_USINT(255.0/100*PwmChannel1);
END_SET
END_PROPERTY

{attribute 'monitoring' := 'call'}
PROPERTY PwmChannel2 : LREAL
GET
PwmChannel2	:= 100.0/255*_stNctProcessDataOut.AppData3;
END_GET
SET
_stNctProcessDataOut.AppData3	:= LREAL_TO_USINT(255.0/100*PwmChannel2);
END_SET
END_PROPERTY

{attribute 'monitoring' := 'call'}
PROPERTY PwmChannel3 : LREAL
GET
PwmChannel3	:= 100.0/255*_stNctProcessDataOut.AppData4;
END_GET
SET
_stNctProcessDataOut.AppData4	:= LREAL_TO_USINT(255.0/100*PwmChannel3);
END_SET
END_PROPERTY

{attribute 'monitoring' := 'call'}
PROPERTY PwmFrequency : LREAL
GET
PwmFrequency	:= 32000.0 + ((128000.0-32000.0)/255.0)*_stNctProcessDataOut.AppData1;
END_GET
SET
IF PwmFrequency <= 32000 THEN
	_stNctProcessDataOut.AppData1	:= 0;
ELSIF PwmFrequency >= 128000 THEN
	_stNctProcessDataOut.AppData1	:= 255;
ELSE
	_stNctProcessDataOut.AppData1	:= LREAL_TO_USINT(((PwmFrequency - 32000.0)/(128000.0-32000.0))*255);
END_IF
END_SET
END_PROPERTY

METHOD ReadRegister : REFERENCE TO ST_ReturnStructure

VAR_INPUT
	bExecute		: BOOL;
	stRegisterType	: NctRegisterType;
END_VAR

VAR_OUTPUT
END_VAR

VAR_INST
	//Case
	nCase	: INT;
	
	//Return
	stReturnStructure	: ST_ReturnStructure;

	//Trigger
	fbRTrig: R_TRIG;
	fbFTrig: F_TRIG;

	//Command
	stNctCommandEntry	: NctCommandEntry;
	stNctCommandInfo	: NctCommandInfo;
	stNctCommandData	: ARRAY[1..256] OF BYTE;
	
	//Timeout	
	fbTimeout	: TON;
	
	//LogMessage
	aLogMessageThrown	: ARRAY[1..4] OF BOOL;
END_VAR	
	
VAR	
	//Command
	stNctReadRegisterCommandArguments	: NctReadRegisterCommandArguments;
	stAbortCommandArguments					: NctAbortCommandArguments;
	nDataCounter							: UDINT;
	
	//Timeout
	tTimeoutTime	: TIME :=T#1S;	//Sets the time for timeout
	
	//LogMessage
	nNumLogMessages	: INT :=4;
	nForCounter		: INT;
END_VAR
fbRTrig(CLK:=bExecute);
fbFTrig(CLK:=bExecute);

//On rising Execute
IF fbRTrig.Q THEN
	//Update return
	stReturnStructure.Done		:= FALSE;
	stReturnStructure.Busy		:= TRUE;
	stReturnStructure.Active	:= FALSE;
	stReturnStructure.Aborted	:= FALSE;
	stReturnStructure.Error		:= FALSE;
	stReturnStructure.ErrorId	:= 0;
	
	//Set case
	nCase:=1;

//On falling Execute
ELSIF fbFTrig.Q THEN
	//Update return
	stReturnStructure.Done		:= FALSE;
	stReturnStructure.Busy		:= FALSE;
	stReturnStructure.Active	:= FALSE;
	stReturnStructure.Aborted	:= FALSE;
	stReturnStructure.Error		:= FALSE;
	stReturnStructure.ErrorId	:= 0;

	//Set case
	nCase:=0;
END_IF

CASE nCase OF
	0: //Idle
		;
	
	1: //Prepare Command
		IF Status.isLocalAddressValid AND Status.isMinActivationTimePassed THEN
		
			//Command Parameters
			stNctReadRegisterCommandArguments.iterationCount		:= 1;
			stNctReadRegisterCommandArguments.maxErrorCount		:= 10;
			stNctReadRegisterCommandArguments.executionMode		:= NctCommandExecutionMode.UntilSuccessMaxErrors;
			stNctReadRegisterCommandArguments.priority			:= 0;
			stNctReadRegisterCommandArguments.registerType		:= stRegisterType;
			stNctReadRegisterCommandArguments.offset				:= 0;
			stNctReadRegisterCommandArguments.size				:= 0;
			
			stNctReadRegisterCommandArguments.options.isResumeOn	:= FALSE;

			//Add Write Init Command
			stNctCommandEntry	:= NctBaseUnitInterface.AddReadRegisterCommand(stNctReadRegisterCommandArguments);
			
			//Update return structure
			stReturnStructure.Done		:= FALSE;
			stReturnStructure.Busy		:= TRUE;
			stReturnStructure.Active	:= FALSE;
			stReturnStructure.Aborted	:= FALSE;
			stReturnStructure.Error		:= FALSE;
			stReturnStructure.ErrorId	:= 0;
			
			//Reset log messages
			FOR nForCounter:=1 TO nNumLogMessages DO
				aLogMessageThrown[nForCounter]	:= FALSE;
			END_FOR
			
			//Reset timeout timer
			fbTimeOut(IN:=FALSE);
			
			//Set case
			nCase:=2;
			
		ELSIF NOT (Status.isLocalAddressValid AND Status.isMinActivationTimePassed) THEN
			//Update return structure
			stReturnStructure.Done		:= FALSE;
			stReturnStructure.Busy		:= FALSE;
			stReturnStructure.Active	:= FALSE;
			stReturnStructure.Aborted	:= FALSE;
			stReturnStructure.Error		:= TRUE;
			stReturnStructure.ErrorId	:= 2;
			
			//Write log message
			IF NOT aLogMessageThrown[stReturnStructure.ErrorId] THEN
				aLogMessageThrown[stReturnStructure.ErrorId]	:= TRUE;
				
				ADSLOGSTR(msgCtrlMask:=ADSLOG_MSGTYPE_ERROR ,msgFmtStr:='Read Register of %s not possible because the Base Unit is not ready to process commands.',strArg:=NctBaseUnitInterface.P_ObjectName);
			END_IF
		
			//Set case
			nCase:=0;
			
		ELSE
			//Update return structure
			stReturnStructure.Done		:= FALSE;
			stReturnStructure.Busy		:= FALSE;
			stReturnStructure.Active	:= FALSE;
			stReturnStructure.Aborted	:= FALSE;
			stReturnStructure.Error		:= TRUE;
			stReturnStructure.ErrorId	:= 1;
			
			//Write log message
			IF NOT aLogMessageThrown[stReturnStructure.ErrorId] THEN
				aLogMessageThrown[stReturnStructure.ErrorId]	:= TRUE;
				
				ADSLOGSTR(msgCtrlMask:=ADSLOG_MSGTYPE_ERROR ,msgFmtStr:='Read Register of %s not possible because of a general Error.',strArg:=NctBaseUnitInterface.P_ObjectName);
			END_IF
			
			//Next step
			nCase:=0;	
			
		END_IF

	2: //Check Command
		stNctCommandInfo	:= NctBaseUnitInterface.GetCmdInfoByCmdEntry(stNctCommandEntry);
	
		IF 		stNctCommandInfo.status = NctCommandStatus.IsRunning THEN
			//Update return structure
			stReturnStructure.Done		:= FALSE;
			stReturnStructure.Busy		:= TRUE;
			stReturnStructure.Active	:= TRUE;
			stReturnStructure.Aborted	:= FALSE;
			stReturnStructure.Error		:= FALSE;
			stReturnStructure.ErrorId	:= 0;
			
			//Timeout
			fbTimeOut(IN:=TRUE, PT:=tTimeoutTime);
			
			IF fbTimeOut.Q THEN
				//Abort Command
				stAbortCommandArguments.option	:= NctAbortCommandParameterOption.ById;
				stAbortCommandArguments.id		:= stNctCommandEntry.id;
				NctBaseUnitInterface.AbortCommand(stAbortCommandArguments);
				
				//Update return structure
				stReturnStructure.Done		:= FALSE;
				stReturnStructure.Busy		:= FALSE;
				stReturnStructure.Active	:= FALSE;
				stReturnStructure.Aborted	:= FALSE;
				stReturnStructure.Error		:= TRUE;
				stReturnStructure.ErrorId	:= 4;
				
				//Write log message
				IF NOT aLogMessageThrown[stReturnStructure.ErrorId] THEN
					aLogMessageThrown[stReturnStructure.ErrorId]	:= TRUE;
					
					ADSLOGSTR(msgCtrlMask:=ADSLOG_MSGTYPE_ERROR ,msgFmtStr:='Reed Register of %s not possible because the method went into timeout.',strArg:=NctBaseUnitInterface.P_ObjectName);
				END_IF
				
				//Next step
				nCase:=0;
			END_IF
			
		ELSIF 	stNctCommandInfo.status = NctCommandStatus.IsQueued OR
				stNctCommandInfo.status = NctCommandStatus.IsWaitingForStartConditions OR
				stNctCommandInfo.status = NctCommandStatus.IsWaitingToResume THEN
				
			//Update return structure
			stReturnStructure.Done		:= FALSE;
			stReturnStructure.Busy		:= TRUE;
			stReturnStructure.Active	:= FALSE;
			stReturnStructure.Aborted	:= FALSE;
			stReturnStructure.Error		:= FALSE;
			stReturnStructure.ErrorId	:= 0;	
			
		ELSIF 	stNctCommandInfo.status = NctCommandStatus.IsSucceeded THEN
			stNctCommandData	:= NctBaseUnitInterface.GetCmdDataByCmdEntry(stNctCommandEntry);
			
			//Process Data
			_stNctProcessDataIn.AppData0	:= stNctCommandData[1];
			_stNctProcessDataIn.AppData1	:= stNctCommandData[2];
			_stNctProcessDataIn.AppData2	:= stNctCommandData[3];
			_stNctProcessDataIn.AppData3	:= stNctCommandData[4];
			_stNctProcessDataIn.AppData4	:= stNctCommandData[5];
			
			
			//Update return structure
			stReturnStructure.Done		:= TRUE;
			stReturnStructure.Busy		:= FALSE;
			stReturnStructure.Active	:= FALSE;
			stReturnStructure.Aborted	:= FALSE;
			stReturnStructure.Error		:= FALSE;
			stReturnStructure.ErrorId	:= 0;
		
			//Next step
			nCase:=0;
			
		ELSIF 	stNctCommandInfo.status = NctCommandStatus.IsAbortedByArea OR
				stNctCommandInfo.status = NctCommandStatus.IsAbortedByUser THEN
				
			//Update return structure
			stReturnStructure.Done		:= FALSE;
			stReturnStructure.Busy		:= FALSE;
			stReturnStructure.Active	:= FALSE;
			stReturnStructure.Aborted	:= TRUE;
			stReturnStructure.Error		:= FALSE;
			stReturnStructure.ErrorId	:= 0;	
				
			//Next step
			nCase:=0;
			
		ELSIF 	stNctCommandInfo.status = NctCommandStatus.IsFailed OR
				stNctCommandInfo.status = NctCommandStatus.IsFailedDueToChildCommand OR
				stNctCommandInfo.status = NctCommandStatus.IsInitFailedDueToCorruptedArgs OR
				stNctCommandInfo.status = NctCommandStatus.IsInitFailedDueToInvalidArgs OR
				stNctCommandInfo.status = NctCommandStatus.IsInitFailedDueToNoMemory OR
				stNctCommandInfo.status = NctCommandStatus.IsInitFailedDueToNotSupportedRegister THEN
				
			//Update return structure
			stReturnStructure.Done		:= FALSE;
			stReturnStructure.Busy		:= FALSE;
			stReturnStructure.Active	:= FALSE;
			stReturnStructure.Aborted	:= FALSE;
			stReturnStructure.Error		:= TRUE;
			stReturnStructure.ErrorId	:= 3;	
			
			//Write log message
			IF NOT aLogMessageThrown[stReturnStructure.ErrorId] THEN
				aLogMessageThrown[stReturnStructure.ErrorId]	:= TRUE;
				
				ADSLOGSTR(msgCtrlMask:=ADSLOG_MSGTYPE_ERROR ,msgFmtStr:='Read Register of %s not possible because command failed.',strArg:=NctBaseUnitInterface.P_ObjectName);
			END_IF
			
			//Next step
			nCase:=0;
			
		ELSIF	stNctCommandInfo.status = NctCommandStatus.NotDefined THEN
			;
		END_IF
			
END_CASE

//Update return structure
ReadRegister	REF= stReturnStructure;
END_METHOD

{attribute 'monitoring' := 'call'}
PROPERTY Status : REFERENCE TO NctBaseUnitStatus
GET
IF IsInterfaceAssigned THEN
	Status REF= _ipTcIoXtsNctBaseUnitInterface.GetStatus();
END_IF
END_GET
END_PROPERTY

METHOD UpdateProcessData : REFERENCE TO ST_ReturnStructure

VAR_INPUT
	bEnable	: BOOL;	//Enables the cylcilc communication
END_VAR

VAR_OUTPUT
END_VAR

VAR_INST
	//Case
	nCase	: INT;
	
	//Command
	stNctCommandEntry	: NctCommandEntry;
	stNctCommandInfo	: NctCommandInfo;
	stNctCommandData	: ARRAY[1..256] OF BYTE;
	
	//Return
	stReturnStructure	: ST_ReturnStructure;
	
	//Timeout	
	fbTimeout	: TON;
	
	//LogMessage
	aLogMessageThrown	: ARRAY[1..4] OF BOOL;
END_VAR	
	
VAR	
	//Command
	stNctUpdateProcessDataCOmmandArguments	: NctUpdateProcessDataCommandArguments;
	stAbortCommandArguments				: NctAbortCommandArguments;

	//Timeout
	tTimeoutTime	: TIME :=T#5S;	//Sets the time for timeout
	
	//LogMessage
	nNumLogMessages	: INT :=4;
	nForCounter		: INT;
END_VAR
CASE nCase OF
	0: //Prepare Command
		//Executes, if data exchange is enabled by user and Base Unit is ready to receive commands
		IF bEnable AND Status.isLocalAddressValid AND Status.isMinActivationTimePassed THEN

			//Command Parameters
			stNctUpdateProcessDataCOmmandArguments.iterationCount		:= 1;
			stNctUpdateProcessDataCOmmandArguments.maxErrorCount		:= 10;
			stNctUpdateProcessDataCOmmandArguments.executionMode		:= NctCommandExecutionMode.UntilSuccess;
			stNctUpdateProcessDataCOmmandArguments.priority				:= 0;
			
			stNctUpdateProcessDataCOmmandArguments.options.isResumeOn	:= FALSE;
			
			//Process Data
			stNctUpdateProcessDataCOmmandArguments.data[0]	:= _stNctProcessDataOut.AppData0;
			stNctUpdateProcessDataCOmmandArguments.data[1]	:= _stNctProcessDataOut.AppData1;
			stNctUpdateProcessDataCOmmandArguments.data[2]	:= _stNctProcessDataOut.AppData2;
			stNctUpdateProcessDataCOmmandArguments.data[3]	:= _stNctProcessDataOut.AppData3;
			stNctUpdateProcessDataCOmmandArguments.data[4]	:= _stNctProcessDataOut.AppData4;
			
			//Add Write Process Data Command
			stNctCommandEntry	:= NctBaseUnitInterface.AddUpdateProcessDataCommand(stNctUpdateProcessDataCOmmandArguments);
			
			//Update return structure
			stReturnStructure.Done		:= FALSE;
			stReturnStructure.Busy		:= TRUE;
			stReturnStructure.Active	:= FALSE;
			stReturnStructure.Aborted	:= FALSE;
			stReturnStructure.Error		:= FALSE;
			stReturnStructure.ErrorId	:= 0;
			
			//Reset log messages
			FOR nForCounter:=1 TO nNumLogMessages DO
				aLogMessageThrown[nForCounter]	:= FALSE;
			END_FOR
			
			//Reset timeout timer
			fbTimeOut(IN:=FALSE);
			
			//Next step
			nCase:=1;
			
		ELSIF bEnable AND NOT (Status.isLocalAddressValid AND Status.isMinActivationTimePassed) THEN
			//Update return
			stReturnStructure.Done		:= FALSE;
			stReturnStructure.Busy		:= FALSE;
			stReturnStructure.Active	:= FALSE;
			stReturnStructure.Aborted	:= FALSE;
			stReturnStructure.Error		:= TRUE;
			stReturnStructure.ErrorId	:= 2;
			
			//Write log message
			IF NOT aLogMessageThrown[stReturnStructure.ErrorId] THEN
				aLogMessageThrown[stReturnStructure.ErrorId]	:= TRUE;
				
				ADSLOGSTR(msgCtrlMask:=ADSLOG_MSGTYPE_ERROR ,msgFmtStr:='Update Process Data of %s not possible because the Base Unit is not ready to process commands.',strArg:=NctBaseUnitInterface.P_ObjectName);
			END_IF
			
			//Next step
			nCase:=0;
		
		ELSIF NOT bEnable THEN
			//Update return structure
			stReturnStructure.Done		:= FALSE;
			stReturnStructure.Busy		:= FALSE;
			stReturnStructure.Active	:= FALSE;
			stReturnStructure.Aborted	:= FALSE;
			stReturnStructure.Error		:= FALSE;
			stReturnStructure.ErrorId	:= 0;
			
			//Reset log messages
			FOR nForCounter:=1 TO nNumLogMessages DO
				aLogMessageThrown[nForCounter]	:= FALSE;
			END_FOR
			
			//Next step
			nCase:=0;
		
		ELSE
			//Update return structure
			stReturnStructure.Done		:= FALSE;
			stReturnStructure.Busy		:= FALSE;
			stReturnStructure.Active	:= FALSE;
			stReturnStructure.Aborted	:= FALSE;
			stReturnStructure.Error		:= TRUE;
			stReturnStructure.ErrorId	:= 1;
			
			//Write log message
			IF NOT aLogMessageThrown[stReturnStructure.ErrorId] THEN
				aLogMessageThrown[stReturnStructure.ErrorId]	:= TRUE;
				
				ADSLOGSTR(msgCtrlMask:=ADSLOG_MSGTYPE_ERROR ,msgFmtStr:='Update Process Data of %s not possible because of a general Error.',strArg:=NctBaseUnitInterface.P_ObjectName);
			END_IF
			
			//Next step
			nCase:=0;	
		END_IF
	
		
	1:	//Check Command
		stNctCommandInfo	:= NctBaseUnitInterface.GetCmdInfoByCmdEntry(stNctCommandEntry);
	
		IF 		stNctCommandInfo.status = NctCommandStatus.IsRunning THEN
			//Update return structure
			stReturnStructure.Done		:= FALSE;
			stReturnStructure.Busy		:= TRUE;
			stReturnStructure.Active	:= TRUE;
			stReturnStructure.Aborted	:= FALSE;
			stReturnStructure.Error		:= FALSE;
			stReturnStructure.ErrorId	:= 0;
			
			//Timeout
			fbTimeOut(IN:=TRUE, PT:=tTimeoutTime);
			
			IF fbTimeOut.Q THEN
				//Abort Command
				stAbortCommandArguments.option	:= NctAbortCommandParameterOption.ById;
				stAbortCommandArguments.id		:= stNctCommandEntry.id;
				NctBaseUnitInterface.AbortCommand(stAbortCommandArguments);
				
				//Update return structure
				stReturnStructure.Done		:= FALSE;
				stReturnStructure.Busy		:= FALSE;
				stReturnStructure.Active	:= FALSE;
				stReturnStructure.Aborted	:= FALSE;
				stReturnStructure.Error		:= TRUE;
				stReturnStructure.ErrorId	:= 4;
				
				//Write log message
				IF NOT aLogMessageThrown[stReturnStructure.ErrorId] THEN
					aLogMessageThrown[stReturnStructure.ErrorId]	:= TRUE;
					
					ADSLOGSTR(msgCtrlMask:=ADSLOG_MSGTYPE_ERROR ,msgFmtStr:='Update Process Data of %s not possible because the method went into timeout.',strArg:=NctBaseUnitInterface.P_ObjectName);
				END_IF
				
				//Next step
				nCase:=0;
			END_IF
			
		ELSIF 	stNctCommandInfo.status = NctCommandStatus.IsQueued OR
				stNctCommandInfo.status = NctCommandStatus.IsWaitingForStartConditions OR
				stNctCommandInfo.status = NctCommandStatus.IsWaitingToResume THEN
				
			//Update return structure
			stReturnStructure.Done		:= FALSE;
			stReturnStructure.Busy		:= TRUE;
			stReturnStructure.Active	:= FALSE;
			stReturnStructure.Aborted	:= FALSE;
			stReturnStructure.Error		:= FALSE;
			stReturnStructure.ErrorId	:= 0;	
			
		ELSIF 	stNctCommandInfo.status = NctCommandStatus.IsSucceeded THEN
			stNctCommandData	:= NctBaseUnitInterface.GetCmdDataByCmdEntry(stNctCommandEntry);
			
			//Process Data
			_stNctProcessDataIn.AppData0	:= stNctCommandData[1];
			_stNctProcessDataIn.AppData1	:= stNctCommandData[2];
			_stNctProcessDataIn.AppData2	:= stNctCommandData[3];
			_stNctProcessDataIn.AppData3	:= stNctCommandData[4];
			_stNctProcessDataIn.AppData4	:= stNctCommandData[5];
			
			//Update return structure
			stReturnStructure.Done		:= TRUE;
			stReturnStructure.Busy		:= FALSE;
			stReturnStructure.Active	:= FALSE;
			stReturnStructure.Aborted	:= FALSE;
			stReturnStructure.Error		:= FALSE;
			stReturnStructure.ErrorId	:= 0;
		
			//Next step
			nCase:=0;
			
		ELSIF 	stNctCommandInfo.status = NctCommandStatus.IsAbortedByArea OR
				stNctCommandInfo.status = NctCommandStatus.IsAbortedByUser THEN
				
			//Update return structure
			stReturnStructure.Done		:= FALSE;
			stReturnStructure.Busy		:= FALSE;
			stReturnStructure.Active	:= FALSE;
			stReturnStructure.Aborted	:= TRUE;
			stReturnStructure.Error		:= FALSE;
			stReturnStructure.ErrorId	:= 0;	
				
			//Next step
			nCase:=0;
			
		ELSIF 	stNctCommandInfo.status = NctCommandStatus.IsFailed OR
				stNctCommandInfo.status = NctCommandStatus.IsFailedDueToChildCommand OR
				stNctCommandInfo.status = NctCommandStatus.IsInitFailedDueToCorruptedArgs OR
				stNctCommandInfo.status = NctCommandStatus.IsInitFailedDueToInvalidArgs OR
				stNctCommandInfo.status = NctCommandStatus.IsInitFailedDueToNoMemory OR
				stNctCommandInfo.status = NctCommandStatus.IsInitFailedDueToNotSupportedRegister THEN
				
			//Update return structure
			stReturnStructure.Done		:= FALSE;
			stReturnStructure.Busy		:= FALSE;
			stReturnStructure.Active	:= FALSE;
			stReturnStructure.Aborted	:= FALSE;
			stReturnStructure.Error		:= TRUE;
			stReturnStructure.ErrorId	:= 3;	
			
			//Write log message
			IF NOT aLogMessageThrown[stReturnStructure.ErrorId] THEN
				aLogMessageThrown[stReturnStructure.ErrorId]	:= TRUE;
				
				ADSLOGSTR(msgCtrlMask:=ADSLOG_MSGTYPE_ERROR ,msgFmtStr:='Update Process Data of %s not possible because command failed.',strArg:=NctBaseUnitInterface.P_ObjectName);
			END_IF
			
			//Next step
			nCase:=0;
			
		ELSIF	stNctCommandInfo.status = NctCommandStatus.NotDefined THEN
			;
		END_IF

END_CASE

//Update return structure
UpdateProcessData	REF= stReturnStructure;
END_METHOD

METHOD WriteRegister : REFERENCE TO ST_ReturnStructure

VAR_INPUT
	bExecute		: BOOL;
	stRegisterType	: NctRegisterType;
END_VAR

VAR_OUTPUT
END_VAR

VAR_INST
	//Case
	nCase	: INT;
	
	//Return
	stReturnStructure	: ST_ReturnStructure;

	//Trigger
	fbRTrig: R_TRIG;
	fbFTrig: F_TRIG;

	//Command
	stNctCommandEntry	: NctCommandEntry;
	stNctCommandInfo	: NctCommandInfo;
	stNctCommandData	: ARRAY[1..256] OF BYTE;
	
	//Timeout	
	fbTimeout	: TON;
	
	//LogMessage
	aLogMessageThrown	: ARRAY[1..4] OF BOOL;
END_VAR	
	
VAR	
	//Command
	stNctWriteRegisterCommandArguments	: NctWriteRegisterCommandArguments;
	stAbortCommandArguments					: NctAbortCommandArguments;
	pTempData								: POINTER TO BYTE;
	nDataCounter							: UDINT;
	nDataSize								: UDINT;
	
	//Timeout
	tTimeoutTime	: TIME :=T#1S;	//Sets the time for timeout
	
	//LogMessage
	nNumLogMessages	: INT :=4;
	nForCounter		: INT;

END_VAR
fbRTrig(CLK:=bExecute);
fbFTrig(CLK:=bExecute);

//On rising Execute
IF fbRTrig.Q THEN
	//Update return
	stReturnStructure.Done		:= FALSE;
	stReturnStructure.Busy		:= TRUE;
	stReturnStructure.Active	:= FALSE;
	stReturnStructure.Aborted	:= FALSE;
	stReturnStructure.Error		:= FALSE;
	stReturnStructure.ErrorId	:= 0;
	
	//Set case
	nCase:=1;

//On falling Execute
ELSIF fbFTrig.Q THEN
	//Update return
	stReturnStructure.Done		:= FALSE;
	stReturnStructure.Busy		:= FALSE;
	stReturnStructure.Active	:= FALSE;
	stReturnStructure.Aborted	:= FALSE;
	stReturnStructure.Error		:= FALSE;
	stReturnStructure.ErrorId	:= 0;

	//Set case
	nCase:=0;
END_IF

CASE nCase OF
	0: //Idle
		;
	
	1: //Prepare Command
		IF Status.isLocalAddressValid AND Status.isMinActivationTimePassed THEN
		
			//Command Parameters
			stNctWriteRegisterCommandArguments.iterationCount		:= 1;
			stNctWriteRegisterCommandArguments.maxErrorCount			:= 10;
			stNctWriteRegisterCommandArguments.executionMode			:= NctCommandExecutionMode.UntilSuccessMaxErrors;
			stNctWriteRegisterCommandArguments.priority				:= 0;
			stNctWriteRegisterCommandArguments.registerType			:= stRegisterType;
			stNctWriteRegisterCommandArguments.offset				:= 0;
			stNctWriteRegisterCommandArguments.size					:= 0;
			
			stNctWriteRegisterCommandArguments.options.isResumeOn	:= FALSE;
			
			//Register Type
			CASE stRegisterType OF
				
				NctRegisterType.Bic						: pTempData:=ADR(_aBIC);
				
				NctRegisterType.ControlVoltage			: pTempData:=ADR(_nControlVoltage);
				
				NctRegisterType.DeviceName				: pTempData:=ADR(_sDeviceName);
				
				NctRegisterType.HardwareVersion			: pTempData:=ADR(_sHardwareversion);
				
				NctRegisterType.Identity				: pTempData:=ADR(_stIdentity);
				
				NctRegisterType.MoverGuid				: pTempData:=ADR(_stMoverGuid);
				
				NctRegisterType.MoverUserName			: pTempData:=ADR(_sMoverUsername);
																					
			END_CASE
			
			//Register Data
			IF pTempData <> 0 THEN
				
				nDataSize	:= NctBaseUnitInterface.GetRegisterParameterSize(stRegisterType := stRegisterType);
				
				IF nDataSize <> 0 THEN
					nDataSize	:= nDataSize-1;
				END_IF
				
				FOR nDataCounter := 0 TO nDataSize DO
					stNctWriteRegisterCommandArguments.data[nDataCounter]	:= pTempData[nDataCounter];
					
				END_FOR
			END_IF
			
			//Add Write Init Command
			stNctCommandEntry	:= NctBaseUnitInterface.AddWriteRegisterCommand(stNctWriteRegisterCommandArguments);
			
			//Update return structure
			stReturnStructure.Done		:= FALSE;
			stReturnStructure.Busy		:= TRUE;
			stReturnStructure.Active	:= FALSE;
			stReturnStructure.Aborted	:= FALSE;
			stReturnStructure.Error		:= FALSE;
			stReturnStructure.ErrorId	:= 0;
			
			//Reset log messages
			FOR nForCounter:=1 TO nNumLogMessages DO
				aLogMessageThrown[nForCounter]	:= FALSE;
			END_FOR
			
			//Reset timeout timer
			fbTimeOut(IN:=FALSE);
			
			//Set case
			nCase:=2;
			
		ELSIF NOT (Status.isLocalAddressValid AND Status.isMinActivationTimePassed) THEN
			//Update return structure
			stReturnStructure.Done		:= FALSE;
			stReturnStructure.Busy		:= FALSE;
			stReturnStructure.Active	:= FALSE;
			stReturnStructure.Aborted	:= FALSE;
			stReturnStructure.Error		:= TRUE;
			stReturnStructure.ErrorId	:= 2;
			
			//Write log message
			IF NOT aLogMessageThrown[stReturnStructure.ErrorId] THEN
				aLogMessageThrown[stReturnStructure.ErrorId]	:= TRUE;
				
				ADSLOGSTR(msgCtrlMask:=ADSLOG_MSGTYPE_ERROR ,msgFmtStr:='Write Register of %s not possible because the Base Unit is not ready to process commands.',strArg:=NctBaseUnitInterface.P_ObjectName);
			END_IF
		
			//Set case
			nCase:=0;
			
		ELSE
			//Update return structure
			stReturnStructure.Done		:= FALSE;
			stReturnStructure.Busy		:= FALSE;
			stReturnStructure.Active	:= FALSE;
			stReturnStructure.Aborted	:= FALSE;
			stReturnStructure.Error		:= TRUE;
			stReturnStructure.ErrorId	:= 1;
			
			//Write log message
			IF NOT aLogMessageThrown[stReturnStructure.ErrorId] THEN
				aLogMessageThrown[stReturnStructure.ErrorId]	:= TRUE;
				
				ADSLOGSTR(msgCtrlMask:=ADSLOG_MSGTYPE_ERROR ,msgFmtStr:='Write Register of %s not possible because of a general Error.',strArg:=NctBaseUnitInterface.P_ObjectName);
			END_IF
			
			//Next step
			nCase:=0;	
			
		END_IF

	2: //Check Command
		stNctCommandInfo	:= NctBaseUnitInterface.GetCmdInfoByCmdEntry(stNctCommandEntry);
	
		IF 		stNctCommandInfo.status = NctCommandStatus.IsRunning THEN
			//Update return structure
			stReturnStructure.Done		:= FALSE;
			stReturnStructure.Busy		:= TRUE;
			stReturnStructure.Active	:= TRUE;
			stReturnStructure.Aborted	:= FALSE;
			stReturnStructure.Error		:= FALSE;
			stReturnStructure.ErrorId	:= 0;
			
			//Timeout
			fbTimeOut(IN:=TRUE, PT:=tTimeoutTime);
			
			IF fbTimeOut.Q THEN
				//Abort Command
				stAbortCommandArguments.option	:= NctAbortCommandParameterOption.ById;
				stAbortCommandArguments.id		:= stNctCommandEntry.id;
				NctBaseUnitInterface.AbortCommand(stAbortCommandArguments);
				
				//Update return structure
				stReturnStructure.Done		:= FALSE;
				stReturnStructure.Busy		:= FALSE;
				stReturnStructure.Active	:= FALSE;
				stReturnStructure.Aborted	:= FALSE;
				stReturnStructure.Error		:= TRUE;
				stReturnStructure.ErrorId	:= 4;
				
				//Write log message
				IF NOT aLogMessageThrown[stReturnStructure.ErrorId] THEN
					aLogMessageThrown[stReturnStructure.ErrorId]	:= TRUE;
					
					ADSLOGSTR(msgCtrlMask:=ADSLOG_MSGTYPE_ERROR ,msgFmtStr:='Write Register of %s not possible because the method went into timeout.',strArg:=NctBaseUnitInterface.P_ObjectName);
				END_IF
				
				//Next step
				nCase:=0;
			END_IF
			
		ELSIF 	stNctCommandInfo.status = NctCommandStatus.IsQueued OR
				stNctCommandInfo.status = NctCommandStatus.IsWaitingForStartConditions OR
				stNctCommandInfo.status = NctCommandStatus.IsWaitingToResume THEN
				
			//Update return structure
			stReturnStructure.Done		:= FALSE;
			stReturnStructure.Busy		:= TRUE;
			stReturnStructure.Active	:= FALSE;
			stReturnStructure.Aborted	:= FALSE;
			stReturnStructure.Error		:= FALSE;
			stReturnStructure.ErrorId	:= 0;	
			
		ELSIF 	stNctCommandInfo.status = NctCommandStatus.IsSucceeded THEN
			stNctCommandData	:= NctBaseUnitInterface.GetCmdDataByCmdEntry(stNctCommandEntry);
			
			//Process Data
			_stNctProcessDataIn.AppData0	:= stNctCommandData[1];
			_stNctProcessDataIn.AppData1	:= stNctCommandData[2];
			_stNctProcessDataIn.AppData2	:= stNctCommandData[3];
			_stNctProcessDataIn.AppData3	:= stNctCommandData[4];
			_stNctProcessDataIn.AppData4	:= stNctCommandData[5];
			
			
			//Update return structure
			stReturnStructure.Done		:= TRUE;
			stReturnStructure.Busy		:= FALSE;
			stReturnStructure.Active	:= FALSE;
			stReturnStructure.Aborted	:= FALSE;
			stReturnStructure.Error		:= FALSE;
			stReturnStructure.ErrorId	:= 0;
		
			//Next step
			nCase:=0;
			
		ELSIF 	stNctCommandInfo.status = NctCommandStatus.IsAbortedByArea OR
				stNctCommandInfo.status = NctCommandStatus.IsAbortedByUser THEN
				
			//Update return structure
			stReturnStructure.Done		:= FALSE;
			stReturnStructure.Busy		:= FALSE;
			stReturnStructure.Active	:= FALSE;
			stReturnStructure.Aborted	:= TRUE;
			stReturnStructure.Error		:= FALSE;
			stReturnStructure.ErrorId	:= 0;	
				
			//Next step
			nCase:=0;
			
		ELSIF 	stNctCommandInfo.status = NctCommandStatus.IsFailed OR
				stNctCommandInfo.status = NctCommandStatus.IsFailedDueToChildCommand OR
				stNctCommandInfo.status = NctCommandStatus.IsInitFailedDueToCorruptedArgs OR
				stNctCommandInfo.status = NctCommandStatus.IsInitFailedDueToInvalidArgs OR
				stNctCommandInfo.status = NctCommandStatus.IsInitFailedDueToNoMemory OR
				stNctCommandInfo.status = NctCommandStatus.IsInitFailedDueToNotSupportedRegister THEN
				
			//Update return structure
			stReturnStructure.Done		:= FALSE;
			stReturnStructure.Busy		:= FALSE;
			stReturnStructure.Active	:= FALSE;
			stReturnStructure.Aborted	:= FALSE;
			stReturnStructure.Error		:= TRUE;
			stReturnStructure.ErrorId	:= 3;	
			
			//Write log message
			IF NOT aLogMessageThrown[stReturnStructure.ErrorId] THEN
				aLogMessageThrown[stReturnStructure.ErrorId]	:= TRUE;
				
				ADSLOGSTR(msgCtrlMask:=ADSLOG_MSGTYPE_ERROR ,msgFmtStr:='Write Register of %s not possible because command failed.',strArg:=NctBaseUnitInterface.P_ObjectName);
			END_IF
			
			//Next step
			nCase:=0;
			
		ELSIF	stNctCommandInfo.status = NctCommandStatus.NotDefined THEN
			;
		END_IF
			
END_CASE

//Update return structure
WriteRegister	REF= stReturnStructure;
END_METHOD

END_FUNCTION_BLOCK

// ---- POUs/Diagnostics/DiagnosticPRG.TcPOU
PROGRAM DiagnosticPRG
VAR

	// Helpful note: issues with this configuration can throw errors that overload the ADS messages. 
	// It's good to set this task to 1ms cycle time, get it working, then set it to higher speed (2ms, 10ms, etc)
	StartFileStream			: BOOL;
	StopFileStream			: BOOL;
	FileStreamRunning		: BOOL;

	FileStreamController	: FB_ALYC_FileStream;



	// Note Generic Constants in XTSDiagnostic Declaration
	// <Num Movers, Num Modules, Num Infeeds>.  Get this information from XPU structure.  Clothoids count as 2 modules.
	XTSDiagnostic	: FB_XTSDiagnostic <10,12,2>;
	(*
	{IF defined(Product_Selector) OR defined(Product_Selector_Sim)}
	XTSDiagnostic	: ARRAY[0..GVL.NUM_XPU - 1] OF FB_XTSDiagnostic <32,14,4>;
	{ELSIF defined(Bottom_Transport) OR defined(Bottom_Transport_Sim)}
	XTSDiagnostic	: ARRAY[0..GVL.NUM_XPU - 1] OF FB_XTSDiagnostic <26,22,6>;
	{ELSIF defined(Side_Transport) OR defined(Side_Transport_Sim)}
	XTSDiagnostic	: ARRAY[0..GVL.NUM_XPU - 1] OF FB_XTSDiagnostic <38,34,6>;
	{ELSIF defined(EPGS) OR defined(EPGS_Sim)}
	XTSDiagnostic	: ARRAY[0..GVL.NUM_XPU - 1] OF FB_XTSDiagnostic <50,58,13>;
	{END_IF}
	*)

	Init			: BOOL;
	i				: INT;
END_VAR

IF NOT Init THEN
	Action_InitDiag();
	Init	:= TRUE;
END_IF

// Tc Analytics File Stream Control
IF StartFileStream THEN
	FileStreamController.Start();
	StartFileStream		:= FALSE;
ELSIF StopFileStream THEN
	FileStreamController.Stop();
	StopFileStream		:= FALSE;
END_IF
FileStreamRunning		:= FileStreamController.bStarted;

// XTS Diagnostics
XTSDiagnostic.Cyclic();

ACTION Action_InitDiag:
XTSDiagnostic.PowerSupplyCount	:= 2;
XTSDiagnostic.rXTS				REF= MAIN.XTS;

// ********************		SYSTEM 1		******************** //
i := 1;
// Infeed 1
XTSDiagnostic.SetModuleInfeedMapping(i, 1, 1);		i := i + 1;
XTSDiagnostic.SetModuleInfeedMapping(i, 1, 2);		i := i + 1;
XTSDiagnostic.SetModuleInfeedMapping(i, 1, 3);		i := i + 1;
XTSDiagnostic.SetModuleInfeedMapping(i, 1, 4);		i := i + 1;
XTSDiagnostic.SetModuleInfeedMapping(i, 1, 5);		i := i + 1;
XTSDiagnostic.SetModuleInfeedMapping(i, 1, 6);		i := i + 1;

// Infeed 2
XTSDiagnostic.SetModuleInfeedMapping(i, 2, 1);		i := i + 1;
XTSDiagnostic.SetModuleInfeedMapping(i, 2, 2);		i := i + 1;
XTSDiagnostic.SetModuleInfeedMapping(i, 2, 3);		i := i + 1;
XTSDiagnostic.SetModuleInfeedMapping(i, 2, 4);		i := i + 1;
XTSDiagnostic.SetModuleInfeedMapping(i, 2, 5);		i := i + 1;
XTSDiagnostic.SetModuleInfeedMapping(i, 2, 6);		i := i + 1;
END_ACTION

END_PROGRAM

// ---- POUs/Diagnostics/XTSDiag/FB_XTSDiagnostic.TcPOU
FUNCTION_BLOCK FB_XTSDiagnostic
VAR_GENERIC CONSTANT
	NUM_MOVERS				: USINT;
	NUM_MODULES				: USINT;
	NUM_INFEEDS				: USINT;
END_VAR
VAR_INPUT
	ai_DCLinkVoltage AT %I* : ARRAY[0..1] OF UDINT;	// Map to EL9576 Brake Chopper Terminal - DC Link Voltage
	PowerSupplyCount		: INT;					// Number of 48V 20amp power supplies on system
	rXTS					: REFERENCE TO FB_XTS<10>;
END_VAR
VAR_OUTPUT
	{attribute 'TcAnalytics'}
	MoverInfo		AT %Q*		: XTSDiag_MoverInfo;
	MoverInfoByObj			: ARRAY[1..NUM_MOVERS] OF XTSDiag_MoverInfo_ByObj;
	{attribute 'TcAnalytics'}
	ModuleInfo		AT %Q*		: XTSDiag_ModuleInfo;
	ModuleInfoByObj			: ARRAY[1..NUM_MODULES] OF XTSDiag_ModuleInfo_ByObj;
	{attribute 'TcAnalytics'}
	InfeedSectionInfo	AT %Q*	: ARRAY[1..NUM_INFEEDS] OF XTSDiag_InfeedSectionInfo;
	{attribute 'TcAnalytics'}
	SystemInfo		AT %Q*		: XTSDiag_SystemInfo;
END_VAR
VAR
	Init					: BOOL;
	XPUId					: INT;
	_ModuleInfeedMapping	: ARRAY[1..NUM_MODULES] OF XTSDiag_ModuleInfeedMapping_typ;
END_VAR

METHOD Cyclic
VAR_INPUT
END_VAR
VAR
	i			: INT;
	j			: INT;
	Infeed		: INT;
	Position	: INT;
	ConfigCheck	: INT; // 0 is ok
END_VAR
// Do nothing if XTS environment not ready
IF NOT rXTS.System.EnvironmentIsReady THEN
	RETURN;

// Write error message if configuration wrong
ELSIF ConfigCheck > 0 THEN
	IF ConfigCheck = 1 THEN
		ConfigCheck	:= 100;
		ADSLOGSTR( ADSLOG_MSGTYPE_ERROR, 'Invalid FB_XTSDiagnostic configuration - NumMovers > MaxNumMovers','');
	ELSIF ConfigCheck = 2 THEN
		ConfigCheck	:= 100;
		ADSLOGSTR( ADSLOG_MSGTYPE_ERROR, 'Invalid FB_XTSDiagnostic configuration - NumModules > MaxNumModules','');
	END_IF

// Initialize FB
ELSIF NOT Init THEN
	IF GVL_XTSDiag.MAX_NUM_MOVERS < NUM_MOVERS		THEN	ConfigCheck := 1; RETURN; END_IF
	IF GVL_XTSDiag.MAX_NUM_MODULES < NUM_MODULES	THEN	ConfigCheck := 2; RETURN; END_IF
	SystemInfo.MoverCount					:= NUM_MOVERS;
	SystemInfo.ModuleCount					:= NUM_MODULES;
	SystemInfo.AvailableContinuousCurrent	:= PowerSupplyCount * 20.0;
	XPUId									:= 1;//rXTS.System.XPUId;
	FOR i := 1 TO NUM_MODULES DO
		GetInfeedPositionByModule(i, Infeed => Infeed, Position => Position);
		InfeedSectionInfo[Infeed].ModuleNumber[Position]	:= i;
		InfeedSectionInfo[Infeed].ModuleCount				:= InfeedSectionInfo[Infeed].ModuleCount + 1;
	END_FOR
	Init	:= TRUE;
END_IF

// ********************		MOVERS		******************** //
SystemInfo.TotalMoverCurrent		:= 0;
FOR i := 1 TO NUM_MOVERS DO
	MoverInfo.FollowingError[i]		:= rXTS.Mover[i].AxisReference.NcToPlc.PosDiff;
	MoverInfo.SetPosition[i]		:= rXTS.Mover[i].TrackInfo.TrackPosition;
	MoverInfo.SetVelocity[i]		:= rXTS.Mover[i].AxisReference.NcToPlc.SetVelo;
	MoverInfo.SetAcceleration[i]	:= rXTS.Mover[i].AxisReference.NcToPlc.SetAcc;
	MoverInfo.SetCurrent[i]			:= rXTS.System.Environment.XpuTcIo(XPUId).MoverTcIo(i).GetSetCurrent();
	MoverInfo.setForce[i]			:= rXTS.System.Environment.XpuTcIo(XPUId).MoverTcIo(i).GetSetForce();
	MoverInfo.Error[i]				:= rXTS.Mover[i].Error;
	MoverInfo.ErrorID[i]			:= rXTS.Mover[i].ErrorID;
	MoverInfo.Ready[i]				:= rXTS.Mover[i].Ready;

	MoverInfoByObj[i].FollowingError	:= MoverInfo.FollowingError[i];
	MoverInfoByObj[i].SetPosition		:= MoverInfo.SetPosition[i];
	MoverInfoByObj[i].SetVelocity		:= MoverInfo.SetVelocity[i];
	MoverInfoByObj[i].SetAcceleration	:= MoverInfo.SetAcceleration[i];
	MoverInfoByObj[i].SetCurrent		:= MoverInfo.SetCurrent[i];
	MoverInfoByObj[i].setForce			:= MoverInfo.setForce[i];
	MoverInfoByObj[i].Error				:= MoverInfo.Error[i];
	MoverInfoByObj[i].ErrorID			:= MoverInfo.ErrorID[i];
	MoverInfoByObj[i].Ready				:= MoverInfo.Ready[i];

	SystemInfo.TotalMoverCurrent	:= SystemInfo.TotalMoverCurrent + MoverInfo.SetCurrent[i];
END_FOR

// ********************		MOTOR MODULES		******************** //
SystemInfo.TotalModuleCurrent					:= 0;
FOR i := 1 TO NUM_MODULES DO
	ModuleInfo.DCLinkVoltage[i]					:= rXTS.System.Environment.XpuTcIo(XPUId).PartTcIo(1).ModuleTcIo(i).GetDCLinkVoltage();
	ModuleInfo.OverallCurrent[i]				:= rXTS.System.Environment.XpuTcIo(XPUId).PartTcIo(1).ModuleTcIo(i).GetOverallCurrent();
	ModuleInfo.MaxOverallCurrentLast500ms[i]	:= rXTS.System.Environment.XpuTcIo(XPUId).PartTcIo(1).ModuleTcIo(i).GetMaxOverallCurrentLast500ms();
	ModuleInfo.PCBTemperatures[i]				:= rXTS.System.Environment.XpuTcIo(XPUId).PartTcIo(1).ModuleTcIo(i).GetPCBTemperatures();
	ModuleInfo.I2TTemperaturesPct[i]			:= rXTS.System.Environment.XpuTcIo(XPUId).PartTcIo(1).ModuleTcIo(i).GetI2TTemperatures();

	ModuleInfoByObj[i].DCLinkVoltage				:= ModuleInfo.DCLinkVoltage[i];
	ModuleInfoByObj[i].OverallCurrent				:= ModuleInfo.OverallCurrent[i];
	ModuleInfoByObj[i].MaxOverallCurrentLast500ms	:= ModuleInfo.MaxOverallCurrentLast500ms[i];
	ModuleInfoByObj[i].PCBTemperatures				:= ModuleInfo.PCBTemperatures[i];
	ModuleInfoByObj[i].I2TTemperaturesPct			:= ModuleInfo.I2TTemperaturesPct[i];

	SystemInfo.TotalModuleCurrent				:= SystemInfo.TotalModuleCurrent + ModuleInfo.OverallCurrent[i];
END_FOR

// ********************		INFEEDS		******************** //
FOR i := 1 TO NUM_MODULES DO
	GetInfeedPositionByModule(i, Infeed => Infeed, Position => Position);
	InfeedSectionInfo[Infeed].DcLinkVoltage[Position]				:= ModuleInfo.DCLinkVoltage[i];
	InfeedSectionInfo[Infeed].ModuleCurrentSummed[Position]			:= ModuleInfo.OverallCurrent[i];
	InfeedSectionInfo[Infeed].MaxOverallCurrentLast500ms[Position]	:= ModuleInfo.MaxOverallCurrentLast500ms[i];
END_FOR
FOR i := 1 TO NUM_INFEEDS DO
	InfeedSectionInfo[i].StartDcLinkVoltage							:= InfeedSectionInfo[i].DcLinkVoltage[1];
	InfeedSectionInfo[i].EndDcLinkVoltage							:= InfeedSectionInfo[i].DcLinkVoltage[InfeedSectionInfo[i].ModuleCount];
	InfeedSectionInfo[i].VoltageDropAcrossCable						:= (ai_DCLinkVoltage[0] / 1000.0) - InfeedSectionInfo[i].StartDcLinkVoltage;
	InfeedSectionInfo[i].VoltageDropAcrossInfeed					:= InfeedSectionInfo[i].StartDcLinkVoltage - InfeedSectionInfo[i].EndDcLinkVoltage;
	InfeedSectionInfo[i].TotalCurrent								:= InfeedSectionInfo[i].ModuleCurrentSummed[1];
	FOR j := InfeedSectionInfo[i].ModuleCount TO 1 BY -1 DO
		IF j <> InfeedSectionInfo[i].ModuleCount THEN				// Skip the first one since there's no downstream current to subtract
			InfeedSectionInfo[i].ModuleCurrentIndivual[Position]	:= InfeedSectionInfo[i].ModuleCurrentSummed[Position] - InfeedSectionInfo[Infeed].ModuleCurrentSummed[Position + 1];
		END_IF
	END_FOR
END_FOR

// ********************		SYSTEM		******************** //
SystemInfo.BusVoltage[0]	:= ai_DCLinkVoltage[0] / 1000.0;	// units in mV from card
SystemInfo.BusVoltage[1]	:= ai_DCLinkVoltage[1] / 1000.0;
IF SystemInfo.AvailableContinuousCurrent > 0 THEN				// Check for div by 0
	SystemInfo.TotalCurrentUsagePct_MoverCalc	:= SystemInfo.TotalMoverCurrent / SystemInfo.AvailableContinuousCurrent;
	SystemInfo.TotalCurrentUsagePct_ModuleCalc	:= SystemInfo.TotalModuleCurrent / SystemInfo.AvailableContinuousCurrent;
END_IF
END_METHOD

METHOD GetInfeedPositionByModule : BOOL
VAR_INPUT
	Module		: INT;
END_VAR
VAR_OUTPUT
	Infeed		: INT;
	Position	: INT;
END_VAR
Infeed		:= _ModuleInfeedMapping[Module].Infeed;
Position	:= _ModuleInfeedMapping[Module].Position;
END_METHOD

METHOD GetModuleByInfeedPosition : INT
VAR_INPUT
	Infeed		: INT;
	Position	: INT;
END_VAR
VAR_OUTPUT
	Module		: INT;
END_VAR
VAR
	i			: INT;
END_VAR
FOR i := 1 TO NUM_MODULES DO
	IF _ModuleInfeedMapping[Module].Infeed = Infeed AND _ModuleInfeedMapping[Module].Position = Position THEN
		Module	:= i;
		EXIT;
	END_IF
END_FOR
END_METHOD

METHOD SetModuleInfeedMapping
VAR_INPUT
	Module		: INT;
	Infeed		: INT;
	Position	: INT;
END_VAR
_ModuleInfeedMapping[Module].Infeed		:= Infeed;
_ModuleInfeedMapping[Module].Position	:= Position;
END_METHOD

END_FUNCTION_BLOCK

// ---- GlobalTextList.TcGTLO
TEXTLIST GlobalTextList
  453 = '%4.0f mm/s'
  237 = '%4.4f'
  183 = '%d'
  517 = 'Disable'
  232 = 'Enable'
  434 = 'High Velocity'
  919 = 'Low Velocity'
  500 = 'Medium Velocity'
  928 = 'Mover Number'
  80 = 'Offset'
  826 = 'Read From CSV'
  646 = 'Set Mover Offset'
  557 = 'Set Nominal'
  393 = 'Start'
  920 = 'Stop'
  964 = 'Teach Mover Offset'
END_TEXTLIST

// ---- VISUs/Controls.TcVIS
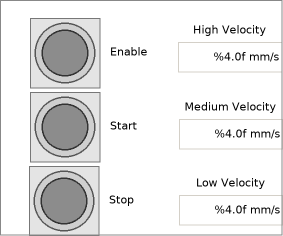
VISUALIZATION Controls  // 283x236
    PushSwitchLed (30,18 70x70), variable: MainCommands.Enable, behaviour: TOGGLE, style: Switch-PushSwitchLed-Gray
    Label (107,37 75x30), "Enable"
    Label (107,111 75x30), "Start"
    PushSwitchLed (30,92 70x70), variable: MainCommands.Start, behaviour: TOGGLE, style: Switch-PushSwitchLed-Gray
    Label (106,185 75x30), "Stop"
    PushSwitchLed (29,166 70x70), variable: MainCommands.Stop, behaviour: TOGGLE, style: Switch-PushSwitchLed-Gray
    Textfield (178,42 104x30), "%4.0f mm/s", text variable: MainCommands.highVelocity
        OnMouseClick: write the text variable via VisuDialogs.Numpad, min 1, max 2000, format %f.0
    Label (181,21 97x18), "High Velocity"
    Textfield (179,119 104x30), "%4.0f mm/s", text variable: MainCommands.mediumVelocity
        OnMouseClick: write the text variable via VisuDialogs.Numpad, min 1, max 2000, format %f.0
    Label (182,98 97x18), "Medium Velocity"
    Textfield (179,195 104x30), "%4.0f mm/s", text variable: MainCommands.lowVelocity
        OnMouseClick: write the text variable via VisuDialogs.Numpad, min 1, max 2000, format %f.0
    Label (182,174 97x18), "Low Velocity"
END_VISUALIZATION
